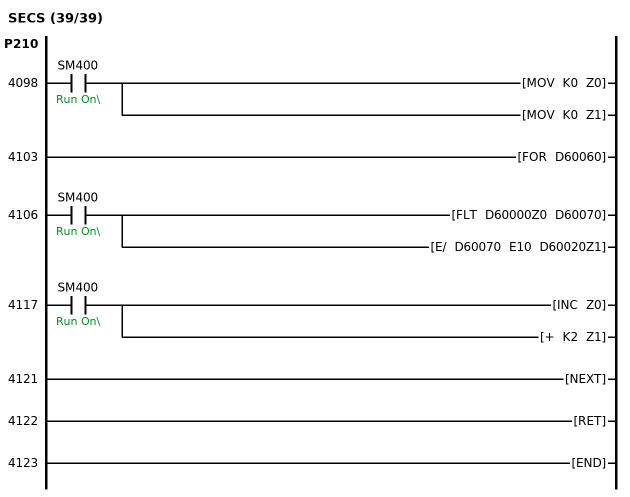
4098  LD      SM400  ; Run On\
      MOV     K0 Z0
      MOV     K0 Z1
4103  FOR     D60060
4106  LD      SM400  ; Run On\
      FLT     D60000Z0 D60070
      E/      D60070 E10 D60020Z1
4117  LD      SM400  ; Run On\
      INC     Z0
      +       K2 Z1
4121  NEXT
4122  RET
4123  END
END_PROGRAM

// device comments not shown above
D5200  ; 溫度到達H01
D5220  ; 溫度到達IRA01
D5240  ; 溫度到達IRB01
D5700  ; 低溫溫度01
D5720  ; 低溫溫度21
D20200  ; A1
D20201  ; B1
X20  ; 進料牙叉上層氣缸上定點
X21  ; 進料牙叉上層氣缸下定點
X22  ; 進料牙叉下層氣缸上定點
X23  ; 進料牙叉下層氣缸下定點
X24  ; 進料牙叉夾板氣缸開定點
X25  ; 進料牙叉夾板氣缸夾定點
X26  ; 進料牙叉左光纖檢知
X27  ; 進料牙叉右光纖檢知
X28  ; 進料吸板真空檢知
X29  ; 進料鼓風機異常
X2A  ; 進料無塵風機異常
X2D  ; 連線_上游出板要求(備用)
X2E  ; 連線_上游出板完成(備用)
X2F  ; 連線_上游備用
X30  ; 進料手臂外氣缸伸出定點
X31  ; 進料手臂外氣缸縮回定點
X32  ; 進料手臂內氣缸伸出定點
X33  ; 進料手臂內氣缸縮回定點
X34  ; 進料手臂上夾板氣缸開定點
X35  ; 進料手臂上夾板氣缸夾定點
X36  ; 進料手臂下夾板氣缸開定點
X37  ; 進料手臂下夾板氣缸夾定點
X38  ; 進料手臂右上有板檢知
X39  ; 進料手臂左上有板檢知
X3A  ; 進料手臂右下有板檢知
X3B  ; 進料手臂左下有板檢知
X3C  ; 進料安全門開關
X3D  ; 進料緊急停止開關
X3E  ; 進/出料蜂鳴器靜音按鈕
X3F  ; 進料氣源壓力檢知
X40  ; 進料回流滿框光電
X41  ; 進料回流檔框1光電
X42  ; 進料回流檔框2光電
X43  ; 進料回流檔框定點光電
X44  ; 進料檔框1氣缸D1上定點
X45  ; 進料檔框1氣缸D1下定點
X46  ; 進料檔框2氣缸D2上定點
X47  ; 進料檔框2氣缸D2下定點
X48  ; 進料後拍框氣缸A13伸出定點
X49  ; 進料後拍框氣缸A13縮回定點
X4A  ; 進料托框氣缸A12上定點
X4B  ; 進料托框氣缸A12下定點
X4C  ; 進料托伸縮氣缸A11A/B伸出定點
X4D  ; 進料托伸縮氣缸A11A/B縮回定點
X4E  ; 進料托框左光電
X4F  ; 進料托框右光電
X50  ; 進料夾框A桿前520光纖
X51  ; 進料夾框A桿前500光纖
X52  ; 進料夾框A桿前260光纖
X53  ; 進料夾框A桿前250光纖
X54  ; 進料夾框B桿前250光纖
X55  ; 進料夾框B桿前260光纖
X56  ; 進料夾框B桿前500光纖
X57  ; 進料夾框B桿前520光纖
X58  ; 進料夾框A桿後520光纖
X59  ; 進料夾框A桿後500光纖
X5A  ; 進料夾框A桿後260光纖
X5B  ; 進料夾框A桿後250光纖
X5C  ; 進料夾框B桿後250光纖
X5D  ; 進料夾框B桿後260光纖
X5E  ; 進料夾框B桿後500光纖
X5F  ; 進料夾框B桿後520光纖
X60  ; 進料左上下夾氣缸A1A/B伸出定點
X61  ; 進料左上下夾氣缸A1A/B縮回定點
X62  ; 進料左拍框氣缸A2伸出定點
X63  ; 進料左拍框氣缸A2縮回定點
X64  ; 進料左背檔框氣缸A3伸出定點
X65  ; 進料左背檔框氣缸A3縮回定點
X66  ; 進料左開爪氣缸A4伸出定點
X67  ; 進料左開爪氣缸A4縮回定點
X68  ; 進料左開框氣缸A5A/B伸出定點
X69  ; 進料左開框氣缸A5A/B縮回定點
X6A  ; 進料左上夾框光電
X6B  ; 進料左上開夾定點光纖
X6C  ; 進料左下開夾定點光纖
X6E  ; 進料左門磁簧開關
X70  ; 進料右上下夾氣缸A1A/B伸出定點
X71  ; 進料右上下夾氣缸A1A/B縮回定點
X72  ; 進料右拍框氣缸A2伸出定點
X73  ; 進料右拍框氣缸A2縮回定點
X74  ; 進料右背檔框氣缸A3伸出定點
X75  ; 進料右背檔框氣缸A3縮回定點
X76  ; 進料右開爪氣缸A4伸出定點
X77  ; 進料右開爪氣缸A4縮回定點
X78  ; 進料右開框氣缸A5A/B伸出定點
X79  ; 進料右開框氣缸A5A/B縮回定點
X7A  ; 進料右上夾框光電
X7B  ; 進料右上開夾定點光纖
X7C  ; 進料右下開夾定點光纖
X7E  ; 進料右門磁簧開關
X80  ; 分流左_伸出氣缸伸出定點
X81  ; 分流左_伸出氣缸縮回定點
X82  ; 分流左_上昇氣缸上定點
X83  ; 分流左_上昇氣缸下定點
X84  ; 分流左_框架上定點光電
X85  ; 分流左_框架下定點光電
X86  ; 分流左_旋轉定點光電
X88  ; 分流右_伸出氣缸伸出定點
X89  ; 分流右_伸出氣缸縮回定點
X8A  ; 分流右_上昇氣缸上定點
X8B  ; 分流右_上昇氣缸下定點
X8C  ; 分流右_框架上定點光電
X8D  ; 分流右_框架下定點光電
X8E  ; 分流右_旋轉定點光電
X90  ; 左IR輸送進框補助氣缸伸出定點
X91  ; 左IR輸送進框補助氣缸縮回定點
X92  ; 左IR輸送進框定位光纖
X93  ; 左IR輸送入口框架光纖
X94  ; 進料輸送排氣風車異常
X95  ; 出料輸送排氣風車異常
X98  ; 右IR輸送進框補助氣缸伸出定點
X99  ; 右IR輸送進框補助氣缸縮回定點
X9A  ; 右IR輸送進框定位光纖
X9B  ; 右IR輸送入口框架光纖
X9C  ; 進料輸送INV-A11運轉
X9D  ; 回流1輸送INV-A1運轉
X9E  ; 回流2輸送INV-A2運轉
X9F  ; 進料分流旋臂馬達INV-A3運轉
X0A0  ; 左IR輸送出框補助氣缸伸出定點
X0A1  ; 左IR輸送出框補助氣缸縮回定點
X0A2  ; 左IR輸送出口框架光纖
X0A3  ; 左IR輸送出框定位光纖
X0A4  ; 左IR輸送出框定點光纖
X0A5  ; 左IR輸送拉框氣缸伸出定點
X0A6  ; 左IR輸送拉框氣缸縮回定點
X0A7  ; 左IR輸送勾框氣缸伸出定點
X0A8  ; 右IR輸送出框補助氣缸伸出定點
X0A9  ; 右IR輸送出框補助氣缸縮回定點
X0AA  ; 右IR輸送出口框架光纖
X0AB  ; 右IR輸送出框定位光纖
X0AC  ; 右IR輸送出框定點光纖
X0AD  ; 右IR輸送拉框氣缸伸出定點
X0AE  ; 右IR輸送拉框氣缸縮回定點
X0AF  ; 右IR輸送勾框氣缸伸出定點
X0B0  ; 合流左_伸出氣缸伸出定點
X0B1  ; 合流左_伸出氣缸縮回定點
X0B2  ; 合流左_上昇氣缸上定點
X0B3  ; 合流左_上昇氣缸下定點
X0B4  ; 合流左_框架上定點光電
X0B5  ; 合流左_框架下定點光電
X0B6  ; 合流左_旋轉定點光電
X0B8  ; 合流右_伸出氣缸伸出定點
X0B9  ; 合流右_伸出氣缸縮回定點
X0BA  ; 合流右_上昇氣缸上定點
X0BB  ; 合流右_上昇氣缸下定點
X0BC  ; 合流右_框架上定點光電
X0BD  ; 合流右_框架下定點光電
X0BE  ; 合流右_旋轉定點光電
X0C0  ; 出料左上下夾氣缸B01A/B伸出定點
X0C1  ; 出料左上下夾氣缸B01A/B縮回定點
X0C2  ; 出料左拍框氣缸B02伸出定點
X0C3  ; 出料左拍框氣缸B02縮回定點
X0C4  ; 出料左背檔框氣缸B03伸出定點
X0C5  ; 出料左背檔框氣缸B03縮回定點
X0C6  ; 出料左開爪氣缸B04伸出定點
X0C7  ; 出料左開爪氣缸B04縮回定點
X0C8  ; 出料左開框氣缸B05A/B伸出定點
X0C9  ; 出料左開框氣缸B05A/B縮回定點
X0CA  ; 出料左上夾框光電
X0CB  ; 出料左上開夾定點光纖
X0CC  ; 出料左下開夾定點光纖
X0CD  ; 出料左無板確認光電
X0CE  ; 出料左門磁簧開關
X0D0  ; 出料右上下夾氣缸B01A/B伸出定點
X0D1  ; 出料右上下夾氣缸B01A/B縮回定點
X0D2  ; 出料右拍框氣缸B02伸出定點
X0D3  ; 出料右拍框氣缸B02縮回定點
X0D4  ; 出料右背檔框氣缸B03伸出定點
X0D5  ; 出料右背檔框氣缸B03縮回定點
X0D6  ; 出料右開爪氣缸B04伸出定點
X0D7  ; 出料右開爪氣缸B04縮回定點
X0D8  ; 出料右開框氣缸B05A/B伸出定點
X0D9  ; 出料右開框氣缸B05A/B縮回定點
X0DA  ; 出料右上夾框光電
X0DB  ; 出料右上開夾定點光纖
X0DC  ; 出料右下開夾定點光纖
X0DD  ; 出料右無板確認光電
X0DE  ; 出料右門磁簧開關
X0E0  ; 出料回流滿框光電
X0E1  ; 出料回流框架檢知光電
X0E2  ; 出料回流框架脫離光電
X0E6  ; 出料下導框氣缸B14伸出定點
X0E7  ; 出料下導框氣缸B14縮回定點
X0E8  ; 出料推框氣缸B13伸出定點
X0E9  ; 出料推框氣缸B13縮回定點
X0EA  ; 出料托框氣缸B12上定點
X0EB  ; 出料托框氣缸B12下一定點
X0EC  ; 出料托框伸縮氣缸B11A/B伸出定點
X0ED  ; 出料托框伸縮氣缸B11A/B縮回定點
X0EE  ; 出料托框左光電
X0EF  ; 出料托框右光電
X0F0  ; 出料手臂外氣缸伸出定點
X0F1  ; 出料手臂外氣缸縮回定點
X0F2  ; 出料手臂內氣缸伸出定點
X0F3  ; 出料手臂內氣缸縮回定點
X0F4  ; 出料手臂上夾板氣缸開定點
X0F5  ; 出料手臂上夾板氣缸夾定點
X0F6  ; 出料手臂下夾板氣缸開定點
X0F7  ; 出料手臂下夾板氣缸夾定點
X0F8  ; 出料手臂右上有板檢知
X0F9  ; 出料手臂左上有板檢知
X0FA  ; 出料手臂右下有板檢知
X0FB  ; 出料手臂左下有板檢知
X0FC  ; 出料安全門開關
X0FD  ; 出料緊急停止開關
X0FE  ; 電源相序檢知
X0FF  ; 出料氣源壓力檢知
X104  ; 出料平台頂昇氣缸上定點
X105  ; 出料平台頂昇氣缸下定點
X106  ; 出料輸送左側光電
X107  ; 出料輸送右側光電
X108  ; 出料輸送入口光電
X109  ; 出料無塵風機異常
X10A  ; 出料旋臂馬達INV-C01運轉
X10B  ; 出料旋臂馬達INV-C02運轉
X10D  ; 連線_下游允許出板
X10E  ; 連線_下游出板中(備用)
X110  ; 左冷卻排氣風車異常
X111  ; 左冷卻無塵風機異常
X112  ; 左IR輸送INV-B01運轉
X118  ; 右冷卻排氣風車異常
X119  ; 右冷卻無塵風機異常
X11A  ; 右IR輸送INV-B01運轉
X11C  ; 第09槽電熱箱H09超溫防止器
X11D  ; 第10槽電熱箱H10超溫防止器
X11E  ; 第11槽電熱箱H11超溫防止器
X11F  ; 第12槽電熱箱H12超溫防止器
X120  ; 第01槽風車馬達過載異常
X121  ; 第02槽風車馬達過載異常
X122  ; 第03槽風車馬達過載異常
X123  ; 第04槽風車馬達過載異常
X124  ; 第05槽風車馬達過載異常
X125  ; 第06槽風車馬達過載異常
X126  ; 第07槽風車馬達過載異常
X127  ; 第08槽風車馬達過載異常
X128  ; 第01槽風車馬達電流檢知
X129  ; 第02槽風車馬達電流檢知
X12A  ; 第03槽風車馬達電流檢知
X12B  ; 第04槽風車馬達電流檢知
X12C  ; 第05槽風車馬達電流檢知
X12D  ; 第06槽風車馬達電流檢知
X12E  ; 第07槽風車馬達電流檢知
X12F  ; 第08槽風車馬達電流檢知
X130  ; 第01槽電熱箱H01超溫防止器
X131  ; 第02槽電熱箱H02超溫防止器
X132  ; 第03槽電熱箱H03超溫防止器
X133  ; 第04槽電熱箱H04超溫防止器
X134  ; 第05槽電熱箱H05超溫防止器
X135  ; 第06槽電熱箱H06超溫防止器
X136  ; 第07槽電熱箱H07超溫防止器
X137  ; 第08槽電熱箱H08超溫防止器
X138  ; 第01槽IR01A超溫防止器
X139  ; 第02槽IR02A超溫防止器
X13A  ; 第03槽IR03A超溫防止器
X13B  ; 第04槽IR04A超溫防止器
X13C  ; 第05槽IR05A超溫防止器
X13D  ; 第06槽IR06A超溫防止器
X13E  ; 第07槽IR07A超溫防止器
X13F  ; 第08槽IR08A超溫防止器
X140  ; 第01槽熱風H01溫度到達
X141  ; 第02槽熱風H02溫度到達
X142  ; 第03槽熱風H03溫度到達
X143  ; 第04槽熱風H04溫度到達
X144  ; 第05槽熱風H05溫度到達
X145  ; 第06槽熱風H06溫度到達
X146  ; 第07槽熱風H07溫度到達
X147  ; 第08槽熱風H08溫度到達
X148  ; 第01槽IR01A溫度到達
X149  ; 第02槽IR02A溫度到達
X14A  ; 第03槽IR03A溫度到達
X14B  ; 第04槽IR04A溫度到達
X14C  ; 第05槽IR05A溫度到達
X14D  ; 第06槽IR06A溫度到達
X14E  ; 第07槽IR07A溫度到達
X14F  ; 第08槽IR08A溫度到達
X150  ; 第01槽H01溫控超溫異常
X151  ; 第02槽H02溫控超溫異常
X152  ; 第03槽H03溫控超溫異常
X153  ; 第04槽H04溫控超溫異常
X154  ; 第05槽H05溫控超溫異常
X155  ; 第06槽H06溫控超溫異常
X156  ; 第07槽H07溫控超溫異常
X157  ; 第08槽H08溫控超溫異常
X158  ; 第01槽IR01A溫控超溫異常
X159  ; 第02槽IR02A溫控超溫異常
X15A  ; 第03槽IR03A溫控超溫異常
X15B  ; 第04槽IR04A溫控超溫異常
X15C  ; 第05槽IR05A溫控超溫異常
X15D  ; 第06槽IR06A溫控超溫異常
X15E  ; 第07槽IR07A溫控超溫異常
X15F  ; 第08槽IR08A溫控超溫異常
X160  ; 第09槽風車馬達過載異常
X161  ; 第10槽風車馬達過載異常
X162  ; 第11槽風車馬達過載異常
X163  ; 第12槽風車馬達過載異常
X164  ; 第09槽風車馬達電流檢知
X165  ; 第10槽風車馬達電流檢知
X166  ; 第11槽風車馬達電流檢知
X167  ; 第12槽風車馬達電流檢知
X168  ; 第09槽SCR09/09A/09B異常
X169  ; 第10槽SCR10/10A/10B異常
X16A  ; 第11槽SCR11/911/11B異常
X16B  ; 第12槽SCR12/12A/12B異常
X16C  ; 第09槽分路開關跳脫異常
X16D  ; 第10槽分路開關跳脫異常
X16E  ; 第11槽分路開關跳脫異常
X16F  ; 第12槽分路開關跳脫異常
X170  ; 第01槽SCR01/01A/01B異常
X171  ; 第02槽SCR02/02A/02B異常
X172  ; 第03槽SCR03/03A/03B異常
X173  ; 第04槽SCR04/04A/04B異常
X174  ; 第05槽SCR05/05A/05B異常
X175  ; 第06槽SCR06/06A/06B異常
X176  ; 第07槽SCR07/07A/07B異常
X177  ; 第08槽SCR08/08A/08B異常
X178  ; 第01槽分路開關跳脫異常
X179  ; 第02槽分路開關跳脫異常
X17A  ; 第03槽分路開關跳脫異常
X17B  ; 第04槽分路開關跳脫異常
X17C  ; 第05槽分路開關跳脫異常
X17D  ; 第06槽分路開關跳脫異常
X17E  ; 第07槽分路開關跳脫異常
X17F  ; 第08槽分路開關跳脫異常
X180  ; 第01槽IR01B溫度到達
X181  ; 第02槽IR02B溫度到達
X182  ; 第03槽IR03B溫度到達
X183  ; 第04槽IR04B溫度到達
X184  ; 第05槽IR05B溫度到達
X185  ; 第06槽IR06B溫度到達
X186  ; 第07槽IR07B溫度到達
X187  ; 第08槽IR08B溫度到達
X188  ; 第01槽IR01B溫控超溫異常
X189  ; 第02槽IR02B溫控超溫異常
X18A  ; 第03槽IR03B溫控超溫異常
X18B  ; 第04槽IR04B溫控超溫異常
X18C  ; 第05槽IR05B溫控超溫異常
X18D  ; 第06槽IR06B溫控超溫異常
X18E  ; 第07槽IR07B溫控超溫異常
X18F  ; 第08槽IR08B溫控超溫異常
X190  ; 第01槽IR01B超溫防止器
X191  ; 第02槽IR02B超溫防止器
X192  ; 第03槽IR03B超溫防止器
X193  ; 第04槽IR04B超溫防止器
X194  ; 第05槽IR05B超溫防止器
X195  ; 第06槽IR06B超溫防止器
X196  ; 第07槽IR07B超溫防止器
X197  ; 第08槽IR08B超溫防止器
X198  ; 第09槽IR09A超溫防止器
X199  ; 第10槽IR10A超溫防止器
X19A  ; 第11槽IR11A超溫防止器
X19B  ; 第12槽IR12A超溫防止器
X19C  ; 第09槽IR09B超溫防止器
X19D  ; 第10槽IR10B超溫防止器
X19E  ; 第11槽IR11B超溫防止器
X19F  ; 第12槽IR12B超溫防止器
X1A0  ; 第09槽熱風H09溫度到達
X1A1  ; 第09槽H09溫控超溫異常
X1A2  ; 第09槽IR09A溫度到達
X1A3  ; 第09槽IR09A溫控超溫異常
X1A4  ; 第09槽IR09B溫度到達
X1A5  ; 第09槽IR09B溫控超溫異常
X1A8  ; 第10槽熱風H10溫度到達
X1A9  ; 第10槽H10溫控超溫異常
X1AA  ; 第10槽IR10A溫度到達
X1AB  ; 第10槽IR10A溫控超溫異常
X1AC  ; 第10槽IR10B溫度到達
X1AD  ; 第10槽IR10B溫控超溫異常
X1B0  ; 第11槽熱風H11溫度到達
X1B1  ; 第11槽H11溫控超溫異常
X1B2  ; 第11槽IR11A溫度到達
X1B3  ; 第11槽IR11A溫控超溫異常
X1B4  ; 第11槽IR11B溫度到達
X1B5  ; 第11槽IR11B溫控超溫異常
X1B8  ; 第12槽熱風H12溫度到達
X1B9  ; 第12槽H12溫控超溫異常
X1BA  ; 第12槽IR12A溫度到達
X1BB  ; 第12槽IR12A溫控超溫異常
X1BC  ; 第12槽IR12B溫度到達
X1BD  ; 第12槽IR12B溫控超溫異常
X0A23  ; Other station   DataLinkStatus
X0A48  ; High resolutuon mode status flag
X0A49  ; Operating condition setting ok
X0A4A  ; Offset/gain setting mode flag
X0A4B  ; Channel change completed flag
X0A4C  ; Set value change completed flag
X0A4D  ; Synchronous mode flag
X1007  ; 進料手臂_(DO08)
X1008  ; 進料手臂_(DO09)
X1009  ; 進料手臂_AB放板#3位置(DO10)
X100D  ; 進料手臂_(DO14)
X1010  ; 進料手臂_(DO17)
X1011  ; 進料手臂_(DO18)
X1012  ; 進料手臂_(DO19)
X1013  ; 進料手臂_(DO20)
X1014  ; 進料手臂_(DO21)
X1015  ; 進料手臂_(DO22)
X1016  ; 進料手臂_(DO23)
X1018  ; 進料手臂_(DO25)
X1019  ; 進料手臂_(DO26)
X101D  ; 進料手臂_(DO30)
X101E  ; 進料手臂_(DO31)
X101F  ; 進料手臂_(DO32)
X1024  ; 進料手臂_CCD再校正一次OK(DO37)
X1026  ; 進料手臂_原點往X軸移動-20MM(DO39
X1027  ; 進料手臂_原點往Y軸移動-20MM(DO40
X1028  ; 進料手臂_原點往T軸正轉移動2度(DO
X1029  ; 進料手臂_(DO42)
X102C  ; 進料手臂_B放板完成位置(DO45)
X102E  ; 進料手臂_(DO47)
X102F  ; 進料手臂_(DO48)
X1030  ; 進料手臂_(DO49)
X1031  ; 進料手臂_(DO50)
X1032  ; 進料手臂_(DO51)
X1033  ; 進料手臂_(DO52)
X1034  ; 進料手臂_(DO53)
X1035  ; 進料手臂_(DO54)
X1036  ; 進料手臂_(DO55)
X1037  ; 進料手臂_(DO56)
X1038  ; 進料手臂_(DO57)
X1039  ; 進料手臂_(DO58)
X103A  ; 進料手臂_(DO59)
X103B  ; 進料手臂_(DO60)
X103C  ; 進料手臂_(DO61)
X103D  ; 進料手臂_(DO62)
X103E  ; 進料手臂_(DO63)
X103F  ; 進料手臂_(DO64)
X1040  ; 進料手臂_放板位置_P32-3(DO65)
X1041  ; 進料手臂_放板位置_P32-2(DO66)
X1042  ; 進料手臂_放板位置_P32-1(DO67)
X1043  ; 進料手臂_放板完成位置_P33-10(DO6
X1044  ; 進料手臂_放板完成位置_P33-9(DO69
X1045  ; 進料手臂_(DO70)
X1046  ; 進料手臂_(DO71)
X1047  ; 進料手臂_(DO72)
X1048  ; 進料手臂_(DO73)
X1049  ; 進料手臂_(DO74)
X104A  ; 進料手臂_(DO75)
X104B  ; 進料手臂_(DO76)
X104C  ; 進料手臂_(DO77)
X104D  ; 進料手臂_(DO78)
X104E  ; 進料手臂_(DO79)
X104F  ; 進料手臂_(DO80)
X1050  ; 進料手臂_(DO81)
X1051  ; 進料手臂_(DO82)
X1052  ; 進料手臂_(DO83)
X1053  ; 進料手臂_(DO84)
X1054  ; 進料手臂_(DO85)
X1055  ; 進料手臂_(DO86)
X1056  ; 進料手臂_(DO87)
X1057  ; 進料手臂_(DO88)
X1058  ; 進料手臂_(DO89)
X1059  ; 進料手臂_(DO90)
X105A  ; 進料手臂_(DO91)
X105B  ; 進料手臂_(DO92)
X105C  ; 進料手臂_(DO93)
X105D  ; 進料手臂_(DO94)
X105E  ; 進料手臂_(DO95)
X105F  ; 進料手臂_(DO96)
X1060  ; 進料手臂_(DO97)
X1061  ; 進料手臂_(DO98)
X1062  ; 進料手臂_(DO99)
X1063  ; 進料手臂_(DO100)
X1064  ; 進料手臂_(DO101)
X1065  ; 進料手臂_(DO102)
X1066  ; 進料手臂_(DO103)
X1067  ; 進料手臂_(DO104)
X1068  ; 進料手臂_(DO105)
X1069  ; 進料手臂_(DO106)
X106A  ; 進料手臂_(DO107)
X106B  ; 進料手臂_(DO108)
X106C  ; 進料手臂_(DO109)
X106D  ; 進料手臂_(DO110)
X106E  ; 進料手臂_(DO111)
X106F  ; 進料手臂_(DO112)
X1070  ; 進料手臂_(DO113)
X1071  ; 進料手臂_(DO114)
X1072  ; 進料手臂_(DO115)
X1073  ; 進料手臂_(DO116)
X1074  ; 進料手臂_(DO117)
X1075  ; 進料手臂_(DO118)
X1076  ; 進料手臂_(DO119)
X1077  ; 進料手臂_(DO120)
X1078  ; 進料手臂_(DO121)
X1079  ; 進料手臂_(DO122)
X107A  ; 進料手臂_(DO123)
X107B  ; 進料手臂_(DO124)
X107C  ; 進料手臂_(DO125)
X107D  ; 進料手臂_(DO126)
X107E  ; 進料手臂_(DO127)
X107F  ; 進料手臂_(DO128)
X1087  ; 出料手臂_(DO08)
X1088  ; 出料手臂_(DO09)
X1089  ; 出料手臂_AB放板#3位置(DO10)
X108D  ; 出料手臂_(DO14)
X1090  ; 出料手臂_(DO17)
X1091  ; 出料手臂_(DO18)
X1092  ; 出料手臂_(DO19)
X1093  ; 出料手臂_(DO20)
X1094  ; 出料手臂_(DO21)
X1095  ; 出料手臂_(DO22)
X1096  ; 出料手臂_(DO23)
X1098  ; 出料手臂_(DO25)
X1099  ; 出料手臂_(DO26)
X109D  ; 出料手臂_(DO30)
X109E  ; 出料手臂_(DO31)
X109F  ; 出料手臂_(DO32)
X10A0  ; 出料手臂_Y+20-OK(DO33)
X10A1  ; 出料手臂_X+20-OK(DO34)
X10A2  ; 出料手臂_Y-20-OK(DO35)
X10A3  ; 出料手臂_X-20-OK(DO36)
X10A4  ; 出料手臂_CCD再校正一次OK(DO37)
X10A5  ; 出料手臂_校正位置OK(DO38)
X10A6  ; 出料手臂_原點往X軸移動-20MM(DO39
X10A7  ; 出料手臂_原點往Y軸移動-20MM(DO40
X10A8  ; 出料手臂_原點往T軸正轉移動2度
X10A9  ; 出料手臂_(DO42)
X10AA  ; 出料手臂_(DO43)
X10AB  ; 出料手臂_B放板上升位置(DO44)
X10AC  ; 出料手臂_B放板完成位置(DO45)
X10AD  ; 出料手臂_T180-OK(DO46)
X10AE  ; 出料手臂_(DO47)
X10AF  ; 出料手臂_(DO48)
X10B0  ; 出料手臂_(DO49)
X10B1  ; 出料手臂_(DO50)
X10B2  ; 出料手臂_(DO51)
X10B3  ; 出料手臂_(DO52)
X10B4  ; 出料手臂_(DO53)
X10B5  ; 出料手臂_(DO54)
X10B6  ; 出料手臂_(DO55)
X10B7  ; 出料手臂_(DO56)
X10B8  ; 出料手臂_(DO57)
X10B9  ; 出料手臂_(DO58)
X10BA  ; 出料手臂_(DO59)
X10BB  ; 出料手臂_(DO60)
X10BC  ; 出料手臂_(DO61)
X10BD  ; 出料手臂_(DO62)
X10BE  ; 出料手臂_(DO63)
X10BF  ; 出料手臂_(DO64)
X10C0  ; 出料手臂_放板位置_P32-3(DO65)
X10C1  ; 出料手臂_放板位置_P32-2(DO66)
X10C2  ; 出料手臂_放板位置_P32-1(DO67)
X10C3  ; 出料手臂_放板完成位置_P33-10(DO6
X10C4  ; 出料手臂_放板完成位置_P33-9(DO69
X10C5  ; 出料手臂_(DO70)
X10C6  ; 出料手臂_(DO71)
X10C7  ; 出料手臂_(DO72)
X10C8  ; 出料手臂_(DO73)
X10C9  ; 出料手臂_(DO74)
X10CA  ; 出料手臂_(DO75)
X10CB  ; 出料手臂_(DO76)
X10CC  ; 出料手臂_(DO77)
X10CD  ; 出料手臂_(DO78)
X10CE  ; 出料手臂_(DO79)
X10CF  ; 出料手臂_(DO80)
X10D0  ; 出料手臂_(DO81)
X10D1  ; 出料手臂_(DO82)
X10D2  ; 出料手臂_(DO83)
X10D3  ; 出料手臂_(DO84)
X10D4  ; 出料手臂_(DO85)
X10D5  ; 出料手臂_(DO86)
X10D6  ; 出料手臂_(DO87)
X10D7  ; 出料手臂_(DO88)
X10D8  ; 出料手臂_(DO89)
X10D9  ; 出料手臂_(DO90)
X10DA  ; 出料手臂_(DO91)
X10DB  ; 出料手臂_(DO92)
X10DC  ; 出料手臂_(DO93)
X10DD  ; 出料手臂_(DO94)
X10DE  ; 出料手臂_(DO95)
X10DF  ; 出料手臂_(DO96)
X10E0  ; 出料手臂_(DO97)
X10E1  ; 出料手臂_(DO98)
X10E2  ; 出料手臂_(DO99)
X10E3  ; 出料手臂_(DO100)
X10E4  ; 出料手臂_(DO101)
X10E5  ; 出料手臂_(DO102)
X10E6  ; 出料手臂_(DO103)
X10E7  ; 出料手臂_(DO104)
X10E8  ; 出料手臂_(DO105)
X10E9  ; 出料手臂_(DO106)
X10EA  ; 出料手臂_(DO107)
X10EB  ; 出料手臂_(DO108)
X10EC  ; 出料手臂_(DO109)
X10ED  ; 出料手臂_(DO110)
X10EE  ; 出料手臂_(DO111)
X10EF  ; 出料手臂_(DO112)
X10F0  ; 出料手臂_(DO113)
X10F1  ; 出料手臂_(DO114)
X10F2  ; 出料手臂_(DO115)
X10F3  ; 出料手臂_(DO116)
X10F4  ; 出料手臂_(DO117)
X10F5  ; 出料手臂_(DO118)
X10F6  ; 出料手臂_(DO119)
X10F7  ; 出料手臂_(DO120)
X10F8  ; 出料手臂_(DO121)
X10F9  ; 出料手臂_(DO122)
X10FA  ; 出料手臂_(DO123)
X10FB  ; 出料手臂_(DO124)
X10FC  ; 出料手臂_(DO125)
X10FD  ; 出料手臂_(DO126)
X10FE  ; 出料手臂_(DO127)
X10FF  ; 出料手臂_(DO128)
Y200  ; 進料牙叉上層氣缸A20上昇SV
Y201  ; 進料牙叉上層氣缸A20下降SV
Y202  ; 進料牙叉下層氣缸A21上昇SV
Y203  ; 進料牙叉下層氣缸A21下降SV
Y204  ; 進料牙叉夾板氣缸A22伸出SV
Y205  ; 進料牙叉夾板氣缸A22縮回SV
Y206  ; 進料真空氣缸A23吸板SV
Y207  ; 進料真空氣缸A23放板SV
Y208  ; 進料真空外側分區A24SV
Y209  ; 進料真空外側分區A25SV
Y20A  ; 進料鼓風機電磁開關
Y20B  ; 進/出料蜂鳴器
Y20C  ; 進/出料三色燈藍燈
Y20D  ; 進/出料三色燈綠燈
Y20E  ; 進/出料三色燈黃燈
Y20F  ; 進/出料三色燈紅燈
Y210  ; 進料手臂板寬氣缸A30伸出SV
Y211  ; 進料手臂板寬氣缸A30縮回SV
Y212  ; 進料手臂上夾板氣缸A31夾板SV
Y213  ; 進料手臂下夾板氣缸A32夾板SV
Y214  ; 進料檔框1氣缸D1伸出SV
Y215  ; 進料檔框1氣缸D1縮回SV
Y216  ; 進料檔框2氣缸D2伸出SV
Y217  ; 進料檔框2氣缸D2縮回SV
Y218  ; 進料後拍框氣缸A13伸出SV
Y219  ; 進料後拍框氣缸A13縮回SV
Y21A  ; 進料托架氣缸A12上昇SV
Y21B  ; 進料托架氣缸A12下降SV
Y21C  ; 進料托框伸縮氣缸伸出SV
Y21D  ; 進料托框伸縮氣缸縮回SV
Y21E  ; CCD照明繼電器
Y220  ; 進料左上下夾框氣缸A1A/B伸出SV
Y221  ; 進料左上下夾框氣缸A1A/B縮回SV
Y222  ; 進料左拍框氣缸A2伸出SV
Y223  ; 進料左拍框氣缸A2縮回SV
Y224  ; 進料左背檔框氣缸A3伸出SV
Y225  ; 進料左背檔框氣缸A3縮回SV
Y226  ; 進料左開爪氣缸A4伸出SV
Y227  ; 進料左開爪氣缸A4縮回SV
Y228  ; 進料左開框氣缸A5A/B伸出SV
Y229  ; 進料左開框氣缸A5A/B縮回SV
Y22D  ; 上游_允許進板訊號
Y22E  ; 上游_進板中訊號
Y22F  ; 上游_啟動完成訊號
Y230  ; 進料右上下夾框氣缸A6A/B伸出SV
Y231  ; 進料右上下夾框氣缸A6A/B縮回SV
Y232  ; 進料右拍框氣缸A7伸出SV
Y233  ; 進料右拍框氣缸A7縮回SV
Y234  ; 進料右背檔框氣缸A8伸出SV
Y235  ; 進料右背檔框氣缸A8縮回SV
Y236  ; 進料右開爪氣缸A9伸出SV
Y237  ; 進料右開爪氣缸A9縮回SV
Y238  ; 進料右開框氣缸A10A/B伸出SV
Y239  ; 進料右開框氣缸A10A/B縮回SV
Y240  ; 分流左_伸出氣缸C1伸出SV
Y241  ; 分流左_伸出氣缸C1縮回SV
Y242  ; 分流左_上昇氣缸C2上昇SV
Y243  ; 分流左_下降氣缸C2下降SV
Y244  ; 左IR輸送進框補助氣缸C3伸出SV
Y245  ; 左IR輸送進框補助氣缸C3縮回SV
Y246  ; 分流右_伸出氣缸C4伸出SV
Y247  ; 分流右_伸出氣缸C4縮回SV
Y248  ; 分流右_上昇氣缸C5上昇SV
Y249  ; 分流右_下降氣缸C5下降SV
Y24A  ; 右IR輸送進框補助氣缸C6伸出SV
Y24B  ; 右IR輸送進框補助氣缸C6縮回SV
Y24C  ; 框架回流輸送1變頻器INVA1運轉
Y24D  ; 框架回流輸送2變頻器INVA2運轉
Y24E  ; 進料分流旋臂變頻器INVA3運轉
Y24F  ; 進料變頻器異常復歸
Y260  ; 合流左_伸出氣缸C11伸出SV
Y261  ; 合流左_伸出氣缸C11縮回SV
Y262  ; 合流左_上昇氣缸C12上昇SV
Y263  ; 合流左_下降氣缸C12下降SV
Y264  ; 左IR輸送出框補助氣缸C13伸出SV
Y265  ; 左IR輸送出框補助氣缸C13縮回SV
Y266  ; 合流右_伸出氣缸C14伸出SV
Y267  ; 合流右_伸出氣缸C14縮回SV
Y268  ; 合流右_上昇氣缸C15上昇SV
Y269  ; 合流右_下降氣缸C15下降SV
Y26A  ; 右IR輸送出框補助氣缸C16伸出SV
Y26B  ; 右IR輸送出框補助氣缸C16縮回SV
Y26C  ; 左IR輸送變頻器INVB1運轉
Y26D  ; 右IR輸送變頻器INVB2運轉
Y26E  ; 出料合流旋臂變頻器INVC1運轉
Y26F  ; 出料變頻器異常復歸
Y270  ; 出料左上下夾框氣缸B1A/B伸出SV
Y271  ; 出料左上下夾框氣缸B1A/B縮回SV
Y272  ; 出料左拍框氣缸B2伸出SV
Y273  ; 出料左拍框氣缸B2縮回SV
Y274  ; 出料左背檔框氣缸B3伸出SV
Y275  ; 出料左背檔框氣缸B3縮回SV
Y276  ; 出料左開爪氣缸B4伸出SV
Y277  ; 出料左開爪氣缸B4縮回SV
Y278  ; 出料左開框氣缸B5A/B伸出SV
Y279  ; 出料左開框氣缸B5A/B縮回SV
Y27A  ; 左IR輸送拉框氣缸C14伸出SV
Y27B  ; 左IR輸送拉框氣缸C14縮回SV
Y27C  ; 左IR輸送勾框氣缸C15伸出SV
Y27D  ; 右IR輸送拉框氣缸C24伸出SV
Y27E  ; 右IR輸送拉框氣缸C24縮回SV
Y27F  ; 右IR輸送勾框氣缸C25伸出SV
Y280  ; 出料右上下夾框氣缸B6A/B伸出SV
Y281  ; 出料右上下夾框氣缸B6A/B縮回SV
Y282  ; 出料右拍框氣缸B7伸出SV
Y283  ; 出料右拍框氣缸B7縮回SV
Y284  ; 出料右背檔框氣缸B8伸出SV
Y285  ; 出料右背檔框氣缸B8縮回SV
Y286  ; 出料右開爪氣缸B9伸出SV
Y287  ; 出料右開爪氣缸B9縮回SV
Y288  ; 出料右開框氣缸B10A/B伸出SV
Y289  ; 出料右開框氣缸B10A/B縮回SV
Y28A  ; 出料平台頂昇氣缸B20上昇SV
Y28B  ; 出料平台頂昇氣缸B20下降SV
Y28D  ; 出料輸送變頻器INVC2運轉
Y28E  ; 出料輸送變頻器INVC2慢速
Y28F  ; 出料輸送變頻器異常復歸
Y290  ; 出料手臂板寬氣缸B30伸出SV
Y291  ; 出料手臂板寬氣缸B30縮回SV
Y292  ; 出料手臂上夾板氣缸B31夾板SV
Y293  ; 出料手臂下夾板氣缸B32夾板SV
Y294  ; 出料下導框氣缸B14伸出SV
Y295  ; 出料下導框氣缸B14縮回SV
Y296  ; 出料推框氣缸B12伸出SV
Y297  ; 出料推框氣缸B12縮回SV
Y298  ; 出料托架氣缸B12上昇SV
Y299  ; 出料托架氣缸B12下降SV
Y29A  ; 出料托框伸縮氣缸B11A/B伸出SV
Y29B  ; 出料托框伸縮氣缸B11A/B縮回SV
Y29D  ; 下游_出板要求訊號
Y29E  ; 下游_出板中訊號
Y29F  ; 下游_啟動完成訊號
Y2A0  ; 第01槽熱風H01電磁開關
Y2A1  ; 第02槽熱風H02電磁開關
Y2A2  ; 第03槽熱風H03電磁開關
Y2A3  ; 第04槽熱風H04電磁開關
Y2A4  ; 第05槽熱風H05電磁開關
Y2A5  ; 第06槽熱風H06電磁開關
Y2A6  ; 第07槽熱風H07電磁開關
Y2A7  ; 第08槽熱風H08電磁開關
Y2A8  ; 第01槽IR01A電磁開關
Y2A9  ; 第02槽IR02A電磁開關
Y2AA  ; 第03槽IR03A電磁開關
Y2AB  ; 第04槽IR04A電磁開關
Y2AC  ; 第05槽IR05A電磁開關
Y2AD  ; 第06槽IR06A電磁開關
Y2AE  ; 第07槽IR07A電磁開關
Y2AF  ; 第08槽IR08A電磁開關
Y2B0  ; 第01槽風車電磁開關
Y2B1  ; 第02槽風車電磁開關
Y2B2  ; 第03槽風車電磁開關
Y2B3  ; 第04槽風車電磁開關
Y2B4  ; 第05槽風車電磁開關
Y2B5  ; 第06槽風車電磁開關
Y2B6  ; 第07槽風車電磁開關
Y2B7  ; 第08槽風車電磁開關
Y2B8  ; 左冷卻排氣風車電磁開關
Y2B9  ; 右冷卻排氣風車電磁開關
Y2BA  ; 進料無塵風機電磁開關
Y2BB  ; 出料無塵風機電磁開關
Y2BC  ; 進料輸送排氣電磁開關
Y2BD  ; 出料輸送排氣電磁開關
Y2BE  ; 左冷卻FFU風機電磁開關
Y2BF  ; 右冷卻FFU風機電磁開關
Y2C0  ; 第09槽熱風H09電磁開關
Y2C1  ; 第10槽熱風H10電磁開關
Y2C2  ; 第11槽熱風H11電磁開關
Y2C3  ; 第12槽熱風H12電磁開關
Y2C8  ; 第09槽IR09A電磁開關
Y2C9  ; 第10槽IR10A電磁開關
Y2CA  ; 第11槽IR11A電磁開關
Y2CB  ; 第12槽IR12A電磁開關
Y2CC  ; 第09槽IR09B電磁開關
Y2CD  ; 第10槽IR10B電磁開關
Y2CE  ; 第11槽IR11B電磁開關
Y2CF  ; 第12槽IR12B電磁開關
Y2D0  ; 第09槽風車電磁開關
Y2D1  ; 第10槽風車電磁開關
Y2D2  ; 第11槽風車電磁開關
Y2D3  ; 第12槽風車電磁開關
Y2D8  ; 第01槽IR01B電磁開關
Y2D9  ; 第02槽IR02B電磁開關
Y2DA  ; 第03槽IR03B電磁開關
Y2DB  ; 第04槽IR04B電磁開關
Y2DC  ; 第05槽IR05B電磁開關
Y2DD  ; 第06槽IR06B電磁開關
Y2DE  ; 第07槽IR07B電磁開關
Y2DF  ; 第08槽IR08B電磁開關
Y0A19  ; #10 AXIS Start
Y0A1F  ; #16 AXIS Start
Y0A43  ; CH03 Output enable/disable flag
Y0A44  ; CH04 Output enable/disable flag
Y0A45  ; CH05 Output enable/disable flag
Y0A46  ; CH06 Output enable/disable flag
Y0A47  ; CH07 Output enable/disable flag
Y0A48  ; CH08 Output enable/disable flag
Y0A49  ; Operating condition setting requ
Y0A4A  ; User range writing request
Y0A4B  ; Channel change request
Y0A4C  ; Set value change request
Y0A4D  ; Synchronous output request
Y1007  ; 進料手臂_(DI08)
Y1008  ; 進料手臂_(DI09)
Y1009  ; 進料手臂_(DI10)
Y100D  ; 進料手臂_(DI14)
Y1011  ; 進料手臂_(DI18)
Y1012  ; 進料手臂_(DI19)
Y1013  ; 進料手臂_(DI20)
Y1015  ; 進料手臂_(DI22)
Y1016  ; 進料手臂_(DI23)
Y1017  ; 進料手臂_(DI24)
Y1018  ; 進料手臂_(DI25)
Y1019  ; 進料手臂_(DI26)
Y101D  ; 進料手臂_(DI30)
Y101E  ; 進料手臂_(DI31)
Y101F  ; 進料手臂_(DI32)
Y1024  ; 進料手臂_CCD再校正一次(DI37)
Y1026  ; 進料手臂_原點往X軸移動-20MM(DI39
Y1027  ; 進料手臂_原點往Y軸移動-20MM(DI40
Y1028  ; 進料手臂_原點往T軸正轉移動2度(DI
Y1029  ; 進料手臂_(DI42)
Y102A  ; 進料手臂_B放板待命位置(DI43)
Y102B  ; 進料手臂_B放板上升位置(DI44)
Y102C  ; 進料手臂_B放板完成位置(DI45)
Y102E  ; 進料手臂_(DI47)
Y102F  ; 進料手臂_(DI48)
Y1030  ; 進料手臂_(DI49)
Y1031  ; 進料手臂_(DI50)
Y1032  ; 進料手臂_(DI51)
Y1033  ; 進料手臂_(DI52)
Y1034  ; 進料手臂_(DI53)
Y1035  ; 進料手臂_(DI54)
Y1036  ; 進料手臂_(DI55)
Y1037  ; 進料手臂_(DI56)
Y1038  ; 進料手臂_(DI57)
Y1039  ; 進料手臂_(DI58)
Y103A  ; 進料手臂_(DI59)
Y103B  ; 進料手臂_(DI60)
Y103C  ; 進料手臂_(DI61)
Y103D  ; 進料手臂_(DI62)
Y103E  ; 進料手臂_(DI63)
Y103F  ; 進料手臂_(DI64)
Y1040  ; 進料手臂_(DI65)
Y1041  ; 進料手臂_(DI66)
Y1042  ; 進料手臂_(DI67)
Y1043  ; 進料手臂_(DI68)
Y1044  ; 進料手臂_(DI69)
Y1045  ; 進料手臂_(DI70)
Y1046  ; 進料手臂_(DI71)
Y1047  ; 進料手臂_(DI72)
Y1048  ; 進料手臂_(DI73)
Y1049  ; 進料手臂_(DI74)
Y104A  ; 進料手臂_(DI75)
Y104B  ; 進料手臂_(DI76)
Y104C  ; 進料手臂_(DI77)
Y104D  ; 進料手臂_(DI78)
Y104E  ; 進料手臂_(DI79)
Y104F  ; 進料手臂_(DI80)
Y1050  ; 進料手臂_(DI81)
Y1051  ; 進料手臂_(DI82)
Y1052  ; 進料手臂_(DI83)
Y1053  ; 進料手臂_(DI84)
Y1054  ; 進料手臂_(DI85)
Y1055  ; 進料手臂_(DI86)
Y1056  ; 進料手臂_(DI87)
Y1057  ; 進料手臂_(DI88)
Y1058  ; 進料手臂_(DI89)
Y1059  ; 進料手臂_(DI90)
Y105A  ; 進料手臂_(DI91)
Y105B  ; 進料手臂_(DI92)
Y105C  ; 進料手臂_(DI93)
Y105D  ; 進料手臂_(DI94)
Y105E  ; 進料手臂_(DI95)
Y105F  ; 進料手臂_(DI96)
Y1060  ; 進料手臂_(DI97)
Y1061  ; 進料手臂_(DI98)
Y1062  ; 進料手臂_(DI99)
Y1063  ; 進料手臂_(DI100)
Y1064  ; 進料手臂_(DI101)
Y1065  ; 進料手臂_(DI102)
Y1066  ; 進料手臂_(DI103)
Y1067  ; 進料手臂_(DI104)
Y1068  ; 進料手臂_(DI105)
Y1069  ; 進料手臂_(DI106)
Y106A  ; 進料手臂_(DI107)
Y106B  ; 進料手臂_(DI108)
Y106C  ; 進料手臂_(DI109)
Y106D  ; 進料手臂_(DI110)
Y106E  ; 進料手臂_(DI111)
Y106F  ; 進料手臂_(DI112)
Y1070  ; 進料手臂_(DI113)
Y1071  ; 進料手臂_(DI114)
Y1072  ; 進料手臂_(DI115)
Y1073  ; 進料手臂_(DI116)
Y1074  ; 進料手臂_(DI117)
Y1075  ; 進料手臂_(DI118)
Y1076  ; 進料手臂_(DI119)
Y1077  ; 進料手臂_(DI120)
Y1078  ; 進料手臂_(DI121)
Y1079  ; 進料手臂_(DI122)
Y107A  ; 進料手臂_(DI123)
Y107B  ; 進料手臂_(DI124)
Y107C  ; 進料手臂_(DI125)
Y107D  ; 進料手臂_(DI126)
Y107E  ; 進料手臂_(DI127)
Y107F  ; 進料手臂_(DI128)
Y1087  ; 出料手臂_(DI08)
Y1088  ; 出料手臂_(DI09)
Y1089  ; 出料手臂_(DI10)
Y108D  ; 出料手臂_(DI14)
Y1091  ; 出料手臂_(DI18)
Y1092  ; 出料手臂_(DI19)
Y1093  ; 出料手臂_(DI20)
Y1095  ; 出料手臂_(DI22)
Y1096  ; 出料手臂_(DI23)
Y1097  ; 出料手臂_(DI24)
Y1098  ; 出料手臂_(DI25)
Y1099  ; 出料手臂_(DI26)
Y109D  ; 出料手臂_(DI30)
Y109E  ; 出料手臂_(DI31)
Y109F  ; 出料手臂_(DI32)
Y10A0  ; 出料手臂_Y+20-GO(DI33)
Y10A1  ; 出料手臂_X+20-GO(DI34)
Y10A2  ; 出料手臂_Y-20(DI35)
Y10A3  ; 出料手臂_X-20(DI36)
Y10A4  ; 出料手臂_CCD再校正一次(DI37)
Y10A5  ; 出料手臂_校正位置IN38(DI38)
Y10A6  ; 出料手臂_原點往X軸移動-20MM(DI39
Y10A7  ; 出料手臂_原點往Y軸移動-20MM(DI40
Y10A8  ; 出料手臂_原點往T軸正轉移動2度
Y10A9  ; 出料手臂_(DI42)
Y10AA  ; 出料手臂_B放板待命位置(DI43)
Y10AB  ; 出料手臂_B放板上升位置(DI44)
Y10AC  ; 出料手臂_B放板完成位置(DI45)
Y10AD  ; 出料手臂_(DI46)
Y10AE  ; 出料手臂_(DI47)
Y10AF  ; 出料手臂_(DI48)
Y10B0  ; 出料手臂_(DI49)
Y10B1  ; 出料手臂_(DI50)
Y10B2  ; 出料手臂_(DI51)
Y10B3  ; 出料手臂_(DI52)
Y10B4  ; 出料手臂_(DI53)
Y10B5  ; 出料手臂_(DI54)
Y10B6  ; 出料手臂_(DI55)
Y10B7  ; 出料手臂_(DI56)
Y10B8  ; 出料手臂_(DI57)
Y10B9  ; 出料手臂_(DI58)
Y10BA  ; 出料手臂_(DI59)
Y10BB  ; 出料手臂_(DI60)
Y10BC  ; 出料手臂_(DI61)
Y10BD  ; 出料手臂_(DI62)
Y10BE  ; 出料手臂_(DI63)
Y10BF  ; 出料手臂_(DI64)
Y10C0  ; 出料手臂_(DI65)
Y10C1  ; 出料手臂_(DI66)
Y10C2  ; 出料手臂_(DI67)
Y10C3  ; 出料手臂_(DI68)
Y10C4  ; 出料手臂_(DI69)
Y10C5  ; 出料手臂_(DI70)
Y10C6  ; 出料手臂_(DI71)
Y10C7  ; 出料手臂_(DI72)
Y10C8  ; 出料手臂_(DI73)
Y10C9  ; 出料手臂_(DI74)
Y10CA  ; 出料手臂_(DI75)
Y10CB  ; 出料手臂_(DI76)
Y10CC  ; 出料手臂_(DI77)
Y10CD  ; 出料手臂_(DI78)
Y10CE  ; 出料手臂_(DI79)
Y10CF  ; 出料手臂_(DI80)
Y10D0  ; 出料手臂_(DI81)
Y10D1  ; 出料手臂_(DI82)
Y10D2  ; 出料手臂_(DI83)
Y10D3  ; 出料手臂_(DI84)
Y10D4  ; 出料手臂_(DI85)
Y10D5  ; 出料手臂_(DI86)
Y10D6  ; 出料手臂_(DI87)
Y10D7  ; 出料手臂_(DI88)
Y10D8  ; 出料手臂_(DI89)
Y10D9  ; 出料手臂_(DI90)
Y10DA  ; 出料手臂_(DI91)
Y10DB  ; 出料手臂_(DI92)
Y10DC  ; 出料手臂_(DI93)
Y10DD  ; 出料手臂_(DI94)
Y10DE  ; 出料手臂_(DI95)
Y10DF  ; 出料手臂_(DI96)
Y10E0  ; 出料手臂_(DI97)
Y10E1  ; 出料手臂_(DI98)
Y10E2  ; 出料手臂_(DI99)
Y10E3  ; 出料手臂_(DI100)
Y10E4  ; 出料手臂_(DI101)
Y10E5  ; 出料手臂_(DI102)
Y10E6  ; 出料手臂_(DI103)
Y10E7  ; 出料手臂_(DI104)
Y10E8  ; 出料手臂_(DI105)
Y10E9  ; 出料手臂_(DI106)
Y10EA  ; 出料手臂_(DI107)
Y10EB  ; 出料手臂_(DI108)
Y10EC  ; 出料手臂_(DI109)
Y10ED  ; 出料手臂_(DI110)
Y10EE  ; 出料手臂_(DI111)
Y10EF  ; 出料手臂_(DI112)
Y10F0  ; 出料手臂_(DI113)
Y10F1  ; 出料手臂_(DI114)
Y10F2  ; 出料手臂_(DI115)
Y10F3  ; 出料手臂_(DI116)
Y10F4  ; 出料手臂_(DI117)
Y10F5  ; 出料手臂_(DI118)
Y10F6  ; 出料手臂_(DI119)
Y10F7  ; 出料手臂_(DI120)
Y10F8  ; 出料手臂_(DI121)
Y10F9  ; 出料手臂_(DI122)
Y10FA  ; 出料手臂_(DI123)
Y10FB  ; 出料手臂_(DI124)
Y10FC  ; 出料手臂_(DI125)
Y10FD  ; 出料手臂_(DI126)
Y10FE  ; 出料手臂_(DI127)
Y10FF  ; 出料手臂_(DI128)
M7  ; 進料輸送停止SW
M14  ; 進料手臂下夾板  夾SW
M15  ; 進料手臂下夾板  放SW
M61  ; 框架回流輸送1   停止SW
M107  ; 出料輸送變頻器停止SW
M161  ; 左IR輸送1   停止SW
M163  ; 右IR輸送2   停止SW
M214  ; 進料手臂下夾板  夾燈
M215  ; 進料手臂下夾板  放燈
M401  ; 1
M402  ; 2
M403  ; 3
M404  ; 4
M512  ; 第13槽  循環風車SW
M513  ; 第14槽  循環風車SW
M514  ; 第15槽  循環風車SW
M515  ; 第16槽  循環風車SW
M516  ; 第17槽  循環風車SW
M517  ; 第18槽  循環風車SW
M518  ; 第19槽  循環風車SW
M519  ; 第20槽  循環風車SW
M550  ; 第01槽  循環風車燈
M551  ; 第02槽  循環風車燈
M552  ; 第03槽  循環風車燈
M553  ; 第04槽  循環風車燈
M554  ; 第05槽  循環風車燈
M555  ; 第06槽  循環風車燈
M556  ; 第07槽  循環風車燈
M557  ; 第08槽  循環風車燈
M558  ; 第09槽  循環風車燈
M559  ; 第10槽  循環風車燈
M560  ; 第11槽  循環風車燈
M561  ; 第12槽  循環風車燈
M562  ; 第13槽  循環風車燈
M563  ; 第14槽  循環風車燈
M564  ; 第15槽  循環風車燈
M565  ; 第16槽  循環風車燈
M566  ; 第17槽  循環風車燈
M567  ; 第18槽  循環風車燈
M568  ; 第19槽  循環風車燈
M569  ; 第20槽  循環風車燈
M580  ; 冷卻排氣左風車燈
M581  ; 冷卻排氣右風車燈
M582  ; 進料無塵風機燈
M583  ; 出料無塵風機燈
M584  ; 進料輸送排氣燈
M585  ; 出料輸送排氣燈
M586  ; 左冷卻  FFU風機 燈
M587  ; 右冷卻  FFU風機 燈
M612  ; 第13槽  電熱SW
M613  ; 第14槽  電熱SW
M614  ; 第15槽  電熱SW
M615  ; 第16槽  電熱SW
M616  ; 第17槽  電熱SW
M617  ; 第18槽  電熱SW
M618  ; 第19槽  電熱SW
M619  ; 第20槽  電熱SW
M650  ; 第01槽  電熱燈
M651  ; 第02槽  電熱燈
M652  ; 第03槽  電熱燈
M653  ; 第04槽  電熱燈
M654  ; 第05槽  電熱燈
M655  ; 第06槽  電熱燈
M656  ; 第07槽  電熱燈
M657  ; 第08槽  電熱燈
M658  ; 第09槽  電熱燈
M659  ; 第10槽  電熱燈
M660  ; 第11槽  電熱燈
M661  ; 第12槽  電熱燈
M662  ; 第13槽  電熱燈
M663  ; 第14槽  電熱燈
M664  ; 第15槽  電熱燈
M665  ; 第16槽  電熱燈
M666  ; 第17槽  電熱燈
M667  ; 第18槽  電熱燈
M668  ; 第19槽  電熱燈
M669  ; 第20槽  電熱燈
M712  ; 第13槽  IRA SW
M713  ; 第14槽  IRA SW
M714  ; 第15槽  IRA SW
M715  ; 第16槽  IRA SW
M716  ; 第17槽  IRA SW
M717  ; 第18槽  IRA SW
M718  ; 第19槽  IRA SW
M719  ; 第20槽  IRA SW
M732  ; 第13槽  IRB SW
M733  ; 第14槽  IRB SW
M734  ; 第15槽  IRB SW
M735  ; 第16槽  IRB SW
M736  ; 第17槽  IRB SW
M737  ; 第18槽  IRB SW
M738  ; 第19槽  IRB SW
M739  ; 第20槽  IRB SW
M750  ; 第01槽  IRA燈
M751  ; 第02槽  IRA燈
M752  ; 第03槽  IRA燈
M753  ; 第04槽  IRA燈
M754  ; 第05槽  IRA燈
M755  ; 第06槽  IRA燈
M756  ; 第07槽  IRA燈
M757  ; 第08槽  IRA燈
M758  ; 第09槽  IRA燈
M759  ; 第10槽  IRA燈
M760  ; 第11槽  IRA燈
M761  ; 第12槽  IRA燈
M762  ; 第13槽  IRA燈
M763  ; 第14槽  IRA燈
M764  ; 第15槽  IRA燈
M765  ; 第16槽  IRA燈
M766  ; 第17槽  IRA燈
M767  ; 第18槽  IRA燈
M768  ; 第19槽  IRA燈
M769  ; 第20槽  IRA燈
M770  ; 第01槽  IRB燈
M771  ; 第02槽  IRB燈
M772  ; 第03槽  IRB燈
M773  ; 第04槽  IRB燈
M774  ; 第05槽  IRB燈
M775  ; 第06槽  IRB燈
M776  ; 第07槽  IRB燈
M777  ; 第08槽  IRB燈
M778  ; 第09槽  IRB燈
M779  ; 第10槽  IRB燈
M780  ; 第11槽  IRB燈
M781  ; 第12槽  IRB燈
M782  ; 第13槽  IRB燈
M783  ; 第14槽  IRB燈
M784  ; 第15槽  IRB燈
M785  ; 第16槽  IRB燈
M786  ; 第17槽  IRB燈
M787  ; 第18槽  IRB燈
M788  ; 第19槽  IRB燈
M789  ; 第20槽  IRB燈
M1002  ; 進料牙叉機構回原點SW
M1012  ; 出料牙叉機構回原點SW
M1013  ; 出料手臂機構回原點SW
M1052  ; 進料牙叉機構回原點燈
M1062  ; 出料牙叉機構回原點燈
M1063  ; 出料手臂機構回原點燈
M1123  ; 進料整板位置04 SW
M1124  ; 進料整板位置05 SW
M1125  ; 進料整板位置06 SW
M1126  ; 進料整板位置07 SW
M1127  ; 進料整板位置08 SW
M1128  ; 進料整板位置09 SW
M1129  ; 進料整板位置10 SW
M1143  ; 進料整板位置04燈
M1144  ; 進料整板位置05燈
M1145  ; 進料整板位置06燈
M1146  ; 進料整板位置07燈
M1147  ; 進料整板位置08燈
M1148  ; 進料整板位置09燈
M1149  ; 進料整板位置10燈
M1222  ; 牙插移載位置03 SW
M1223  ; 牙插移載位置04 SW
M1224  ; 牙插移載位置05 SW
M1225  ; 牙插移載位置06 SW
M1226  ; 牙插移載位置07 SW
M1227  ; 牙插移載位置08 SW
M1228  ; 牙插移載位置09 SW
M1229  ; 牙插移載位置10 SW
M1242  ; 牙插移載位置03燈
M1243  ; 牙插移載位置04燈
M1244  ; 牙插移載位置05燈
M1245  ; 牙插移載位置06燈
M1246  ; 牙插移載位置07燈
M1247  ; 牙插移載位置08燈
M1248  ; 牙插移載位置09燈
M1249  ; 牙插移載位置10燈
M1422  ; 進手臂取手位置03 SW
M1423  ; 進手臂取手位置04 SW
M1424  ; 進手臂取手位置05 SW
M1425  ; 進手臂取手位置06 SW
M1426  ; 進手臂取手位置07 SW
M1427  ; 進手臂取手位置08 SW
M1428  ; 進手臂取手位置09 SW
M1429  ; 進手臂取手位置10 SW
M1442  ; 進手臂取手位置03燈
M1443  ; 進手臂取手位置04燈
M1444  ; 進手臂取手位置05燈
M1445  ; 進手臂取手位置06燈
M1446  ; 進手臂取手位置07燈
M1447  ; 進手臂取手位置08燈
M1448  ; 進手臂取手位置09燈
M1449  ; 進手臂取手位置10燈
M1524  ; 進料托框昇降位置05 SW
M1525  ; 進料托框昇降位置06 SW
M1526  ; 進料托框昇降位置07 SW
M1527  ; 進料托框昇降位置08 SW
M1528  ; 進料托框昇降位置09 SW
M1529  ; 進料托框昇降位置10 SW
M1544  ; 進料托框昇降位置05燈
M1545  ; 進料托框昇降位置06燈
M1546  ; 進料托框昇降位置07燈
M1547  ; 進料托框昇降位置08燈
M1548  ; 進料托框昇降位置09燈
M1549  ; 進料托框昇降位置10燈
M1550  ; 進料托框昇降位置01 SW*
M1551  ; 進料托框昇降位置02 SW*
M1552  ; 進料托框昇降位置03 SW*
M1553  ; 進料托框昇降位置04 SW*
M1554  ; 進料托框昇降位置05 SW*
M1555  ; 進料托框昇降位置06 SW*
M1556  ; 進料托框昇降位置07 SW*
M1557  ; 進料托框昇降位置08 SW*
M1558  ; 進料托框昇降位置09 SW*
M1559  ; 進料托框昇降位置10 SW*
M1625  ; 進左開爪位置06 SW
M1626  ; 進左開爪位置07 SW
M1627  ; 進左開爪位置08 SW
M1628  ; 進左開爪位置09 SW
M1629  ; 進左開爪位置10 SW
M1645  ; 進左開爪位置06燈
M1646  ; 進左開爪位置07燈
M1647  ; 進左開爪位置08燈
M1648  ; 進左開爪位置09燈
M1649  ; 進左開爪位置10燈
M1725  ; 進右開爪位置06 SW
M1726  ; 進右開爪位置07 SW
M1727  ; 進右開爪位置08 SW
M1728  ; 進右開爪位置09 SW
M1729  ; 進右開爪位置10 SW
M1745  ; 進右開爪位置06燈
M1746  ; 進右開爪位置07燈
M1747  ; 進右開爪位置08燈
M1749  ; 進右開爪位置10燈
M1829  ; CCD_HeartBeat心跳
M1857  ; 進料牙叉上昇位置
M1858  ; 進料牙叉下降位置
M1860  ; CCD 對位逾時計次到達
M1873  ; CCD 重置PB
M1875  ; 品種切換PB
M1881  ; CCD基準位置登錄燈
M1883  ; CCD重置燈
M1884  ; Y+20
M1885  ; X-20
M1886  ; Y-20
M1890  ; CCD 重置PLS
M1891  ; 搜索OK  完成
M1892  ; 發生搜索錯誤
M1895  ; 搜索結束PLS
M1897  ; 出料主傳動有板燈
M2123  ; 分流前取框位置04 SW
M2124  ; 分流前取框位置05 SW
M2125  ; 分流前取框位置06 SW
M2126  ; 分流前取框位置07 SW
M2127  ; 分流前取框位置08 SW
M2128  ; 分流前取框位置09 SW
M2129  ; 分流前取框位置10 SW
M2143  ; 分流前取框位置04燈
M2144  ; 分流前取框位置05燈
M2145  ; 分流前取框位置06燈
M2146  ; 分流前取框位置07燈
M2147  ; 分流前取框位置08燈
M2148  ; 分流前取框位置09燈
M2149  ; 分流前取框位置10燈
M2223  ; 合流後掛框位置04 SW
M2224  ; 合流後掛框位置05 SW
M2225  ; 合流後掛框位置06 SW
M2226  ; 合流後掛框位置07 SW
M2227  ; 合流後掛框位置08 SW
M2228  ; 合流後掛框位置09 SW
M2229  ; 合流後掛框位置10 SW
M2243  ; 合流後掛框位置04燈
M2244  ; 合流後掛框位置05燈
M2245  ; 合流後掛框位置06燈
M2246  ; 合流後掛框位置07燈
M2247  ; 合流後掛框位置08燈
M2248  ; 合流後掛框位置09燈
M2249  ; 合流後掛框位置10燈
M2256  ; 出料平台位置07 SW*
M2257  ; 出料平台位置08 SW*
M2258  ; 出料平台位置09 SW*
M2259  ; 出料平台位置10 SW*
M3123  ; 出手臂取手位置04 SW
M3124  ; 出手臂取手位置05 SW
M3125  ; 出手臂取手位置06 SW
M3126  ; 出手臂取手位置07 SW
M3127  ; 出手臂取手位置08 SW
M3128  ; 出手臂取手位置09 SW
M3129  ; 出手臂取手位置10 SW
M3143  ; 出手臂取手位置04燈
M3144  ; 出手臂取手位置05燈
M3145  ; 出手臂取手位置06燈
M3146  ; 出手臂取手位置07燈
M3147  ; 出手臂取手位置08燈
M3148  ; 出手臂取手位置09燈
M3149  ; 出手臂取手位置10燈
M3225  ; 出料托框昇降位置06 SW
M3226  ; 出料托框昇降位置07 SW
M3227  ; 出料托框昇降位置08 SW
M3228  ; 出料托框昇降位置09 SW
M3229  ; 出料托框昇降位置10 SW
M3245  ; 出料托框昇降位置06燈
M3246  ; 出料托框昇降位置07燈
M3247  ; 出料托框昇降位置08燈
M3248  ; 出料托框昇降位置09燈
M3249  ; 出料托框昇降位置10燈
M3325  ; 出左開夾位置06 SW
M3326  ; 出左開夾位置07 SW
M3327  ; 出左開夾位置08 SW
M3328  ; 出左開夾位置09 SW
M3329  ; 出左開夾位置10 SW
M3345  ; 出左開夾位置06燈
M3346  ; 出左開夾位置07燈
M3347  ; 出左開夾位置08燈
M3348  ; 出左開夾位置09燈
M3349  ; 出左開夾位置10燈
M3353  ; 旋轉位置04 SW*
M3354  ; 旋轉位置05 SW*
M3355  ; 旋轉位置06 SW*
M3356  ; 旋轉位置07 SW*
M3357  ; 旋轉位置08 SW*
M3358  ; 旋轉位置09 SW*
M3359  ; 旋轉位置10 SW*
M3425  ; 出右開夾位置06 SW
M3426  ; 出右開夾位置07 SW
M3427  ; 出右開夾位置08 SW
M3428  ; 出右開夾位置09 SW
M3429  ; 出右開夾位置10 SW
M3445  ; 出右開夾位置06燈
M3446  ; 出右開夾位置07燈
M3447  ; 出右開夾位置08燈
M3448  ; 出右開夾位置09燈
M3449  ; 出右開夾位置10燈
M3523  ; 出板牙插移載位置04 SW
M3524  ; 出板牙插移載位置05 SW
M3525  ; 出板牙插移載位置06 SW
M3526  ; 出板牙插移載位置07 SW
M3527  ; 出板牙插移載位置08 SW
M3528  ; 出板牙插移載位置09 SW
M3529  ; 出板牙插移載位置10 SW
M3543  ; 出板牙插移載位置04燈
M3544  ; 出板牙插移載位置05燈
M3545  ; 出板牙插移載位置06燈
M3546  ; 出板牙插移載位置07燈
M3547  ; 出板牙插移載位置08燈
M3548  ; 出板牙插移載位置09燈
M3549  ; 出板牙插移載位置10燈
M4058  ; 預留正極限異常
M4059  ; 預留負極限異常
M4070  ; 預留正極限異常
M4071  ; 預留負極限異常
M4149  ; 進料輸送減速光電異常
M4209  ; 合流右_旋轉定點異常
M4301  ; 第02槽   OTP超溫
M4302  ; 第03槽   OTP超溫
M4303  ; 第04槽   OTP超溫
M4304  ; 第05槽   OTP超溫
M4305  ; 第06槽   OTP超溫
M4306  ; 第07槽   OTP超溫
M4307  ; 第08槽   OTP超溫
M4321  ; 第02槽  IRA OTP 超溫
M4322  ; 第03槽  IRA OTP 超溫
M4323  ; 第04槽  IRA OTP 超溫
M4324  ; 第05槽  IRA OTP 超溫
M4325  ; 第06槽  IRA OTP 超溫
M4326  ; 第07槽  IRA OTP 超溫
M4327  ; 第08槽  IRA OTP 超溫
M4341  ; 第02槽  IRB OTP 超溫
M4342  ; 第03槽  IRB OTP 超溫
M4343  ; 第04槽  IRB OTP 超溫
M4344  ; 第05槽  IRB OTP 超溫
M4345  ; 第06槽  IRB OTP 超溫
M4346  ; 第07槽  IRB OTP 超溫
M4351  ; 第12槽  IRB OTP 超溫
M4421  ; 第02槽 熱風低溫異常
M4422  ; 第03槽 熱風低溫異常
M4423  ; 第04槽 熱風低溫異常
M4424  ; 第05槽 熱風低溫異常
M4425  ; 第06槽 熱風低溫異常
M4426  ; 第07槽 熱風低溫異常
M4427  ; 第08槽 熱風低溫異常
M4428  ; 第09槽 熱風低溫異常
M4429  ; 第10槽 熱風低溫異常
M4430  ; 第11槽 熱風低溫異常
M4431  ; 第12槽 熱風低溫異常
M4441  ; 第02槽 IRA 低溫異常
M4442  ; 第03槽 IRA 低溫異常
M4443  ; 第04槽 IRA 低溫異常
M4444  ; 第05槽 IRA 低溫異常
M4445  ; 第06槽 IRA 低溫異常
M4446  ; 第07槽 IRA 低溫異常
M4447  ; 第08槽 IRA 低溫異常
M4448  ; 第09槽 IRA 低溫異常
M4449  ; 第10槽 IRA 低溫異常
M4450  ; 第11槽 IRA 低溫異常
M4451  ; 第12槽 IRA 低溫異常
M4461  ; 第02槽 IRB 低溫異常
M4462  ; 第03槽 IRB 低溫異常
M4463  ; 第04槽 IRB 低溫異常
M4464  ; 第05槽 IRB 低溫異常
M4465  ; 第06槽 IRB 低溫異常
M4466  ; 第07槽 IRB 低溫異常
M4467  ; 第08槽 IRB 低溫異常
M4468  ; 第09槽 IRB 低溫異常
M4469  ; 第10槽 IRB 低溫異常
M4470  ; 第11槽 IRB 低溫異常
M4471  ; 第12槽 IRB 低溫異常
M4481  ; 第02槽 熱風超溫異常
M4482  ; 第03槽 熱風超溫異常
M4483  ; 第04槽 熱風超溫異常
M4484  ; 第05槽 熱風超溫異常
M4485  ; 第06槽 熱風超溫異常
M4486  ; 第07槽 熱風超溫異常
M4487  ; 第08槽 熱風超溫異常
M4501  ; 第2槽 IRA 超溫異常
M4502  ; 第3槽 IRA 超溫異常
M4503  ; 第4槽 IRA 超溫異常
M4504  ; 第5槽 IRA 超溫異常
M4505  ; 第6槽 IRA 超溫異常
M4506  ; 第7槽 IRA 超溫異常
M4507  ; 第8槽 IRA 超溫異常
M4512  ; 第13槽 IRA 超溫異常
M4513  ; 第14槽 IRA 超溫異常
M4514  ; 第15槽 IRA 超溫異常
M4515  ; 第16槽 IRA 超溫異常
M4521  ; 第2槽 IRB 超溫異常
M4522  ; 第3槽 IRB 超溫異常
M4523  ; 第4槽 IRB 超溫異常
M4524  ; 第5槽 IRB 超溫異常
M4525  ; 第6槽 IRB 超溫異常
M4526  ; 第7槽 IRB 超溫異常
M4527  ; 第8槽 IRB 超溫異常
M4532  ; 第13槽 IRB 超溫異常
M4533  ; 第14槽 IRB 超溫異常
M4534  ; 第15槽 IRB 超溫異常
M4535  ; 第16槽 IRB 超溫異常
M4621  ; 取板牙插驅動器電池異常
M4623  ; 進料手臂取手驅動器電池異常
M4624  ; 進料托框昇降驅動器電池異常
M4625  ; 進左開夾驅動器電池異常
M4626  ; 進右開夾驅動器電池異常
M4630  ; 出料手臂取手驅動器電池異常
M4631  ; 出料托框昇降驅動器電池異常
M4632  ; 出左開夾驅動器電池異常
M4633  ; 出右開夾驅動器電池異常
M4681  ; 取板牙插歸零要求異常
M4683  ; 進料手臂取手歸零要求異常
M4684  ; 進料托框昇降歸零要求異常
M4685  ; 進左開夾歸零要求異常
M4686  ; 進右開夾歸零要求異常
M4687  ; 分流前取框歸零要求異常
M4688  ; 出板牙插歸零要求異常
M4690  ; 出料手臂取手歸零要求異常
M4691  ; 出料托框昇降歸零要求異常
M4692  ; 出左開夾歸零要求異常
M4693  ; 出右開夾歸零要求異常
M4694  ; 合流後掛框歸零要求異常
M4744  ; 印刷機左圍籬安全門偵測ˋ異常
M4745  ; 印刷機右圍籬安全門偵測ˋ異常
M4920  ; 入口計數自保持
M4934  ; 上位允許放板START
M4943  ; 上位下GO_REMOTE
M4944  ; 上位下GO-LOCAL
M5130  ; 回上位面板#1入板訊號
M5135  ; 回上位Panel#1出板訊號
M5150  ; 進料板材尺寸連線模式燈
M5151  ; 出料板材尺寸連線模式燈
M5200  ; 進料I/O測試
M5201  ; 進料I/O 測試_01
M5202  ; 進料I/O 測試_02
M5203  ; 進料I/O 測試_03
M5204  ; 進料I/O 測試_04
M5205  ; 進料I/O 測試_05
M5206  ; 進料I/O 測試_06
M5207  ; 進料I/O 測試_07
M5208  ; 進料I/O 測試_08
M5209  ; 進料I/O 測試_09
M5210  ; 進料I/O 測試_10
M5211  ; 進料I/O 測試_11
M5212  ; 進料I/O 測試_12
M5213  ; 進料I/O 測試_13
M5214  ; 進料I/O 測試_14
M5215  ; 進料I/O 測試_15
M5216  ; 進料I/O 測試_16
M5220  ; 出料I/O測試
M5221  ; 出料I/O 測試_01
M5222  ; 出料I/O 測試_02
M5223  ; 出料I/O 測試_03
M5224  ; 出料I/O 測試_04
M5225  ; 出料I/O 測試_05
M5226  ; 出料I/O 測試_06
M5227  ; 出料I/O 測試_07
M5228  ; 出料I/O 測試_08
M5229  ; 出料I/O 測試_09
M5230  ; 出料I/O 測試_10
M5231  ; 出料I/O 測試_11
M5232  ; 出料I/O 測試_12
M5233  ; 出料I/O 測試_13
M5234  ; 出料I/O 測試_14
M5235  ; 出料I/O 測試_15
M5236  ; 出料I/O 測試_16
M5320  ; FX機台狀態改變
M5410  ; 出料手臂至校正位置手動
M5422  ; 出料手臂自動取板等待點動作條件
M5502  ; PC->Start command
M5503  ; PC->Stop command
M5507  ; 進料開爪位置有板BF
M5508  ; 進料入爐有板BF
M5510  ; 機台狀態BF
M5511  ; 機台狀態INIT
M5512  ; 機台狀態Idle
M5513  ; 機台狀態Ready
M5514  ; 機台狀態Warmup
M5515  ; 機台狀態Exccuting
M5516  ; 機台狀態Pause
M5517  ; 機台狀態Maintenance
M5520  ; 進料段ALARM
M5521  ; 進料段有料
M5522  ; 進料段MOVING
M5523  ; 爐體段ALARM
M5524  ; 爐體段有料
M5525  ; 出料段ALARM
M5526  ; 出料段有料
M5527  ; 出料段MOVING
M5528  ; 回流段ALARM
M5530  ; 機台內有板
M5532  ; 機台LOT生產完畢KP
M6059  ; Host刪除配方
M6060  ; Host刪除配方完成
M6105  ; 回上位新增配方
M6106  ; 回上位刪除配方
M6134  ; 三色燈狀態改變
M6137  ; 手動
M6140  ; 要求上位回讀工單板號右爐
M6141  ; 要求上位回讀工單右爐
M6142  ; 三色黃燈
M6218  ; 和上位連線中
M7017  ; 配方切換旗標
M7022  ; 配方搜尋比對OK
M7026  ; 去空白KP
M7030  ; 配方寫入-KP
M7031  ; 配方寫入-KP
M7035  ; 配方空白
M7040  ; 入口計數自保持
M7042  ; 回上位面板#1入板訊號
M7043  ; 回上位Panel#1出板訊號
M7075  ; 批數歸零旗標
M7076  ; 爐內片數歸零PB
M7077  ; 批次數量歸零PB
M7084  ; TEST
M7120  ; 比對GO-REMOTE字串不對
M7121  ; 名稱GO-LOCAL比對不對
M7122  ; 比對RESUME字串不對
M7123  ; 比對PPID字串不對
M7124  ; 比對PAUSE字串不對
M7125  ; 比對START字串不對
M7126  ; 比對STOP字串不對
M7127  ; 比對PP_SELECT字串不對
M7142  ; [HH-02] 配方搜尋比對NG
M7170  ; [PPID]  配方搜尋比對OK_配方可
M7203  ; 未知?測試用
M7207  ; 上位切換成GO-REMOTE
M7208  ; 上位切換成GO-LOCAL
M7214  ; SECS上位下指令觸發Cmd-燈號
M7322  ; 程式結束
M7604  ; ALARM   暫停
M7605  ; 進料回流光纖暫停
L14  ; 允許進料手臂下夾板  夾
L15  ; 允許進料手臂下夾板  放
L100  ; 停電保持SECS    手動/自動連線
L201  ; Disable Check   FrameL/D
L202  ; Disable Check   SEN. L/D
L203  ; Disable Check   FrameU/D
L204  ; Disable Check   SEN. U/D
L205  ; Disable Check   FrameR/F
L206  ; Disable Check   SEN. R/F
L226  ; 進料牙叉吸風使用
L251  ; 夾爪彈簧偵測
L512  ; 第13槽  循環風車SW  PLS
L513  ; 第14槽  循環風車SW  PLS
L514  ; 第15槽  循環風車SW  PLS
L515  ; 第16槽  循環風車SW  PLS
L516  ; 第17槽  循環風車SW  PLS
L517  ; 第18槽  循環風車SW  PLS
L518  ; 第19槽  循環風車SW  PLS
L519  ; 第20槽  循環風車SW  PLS
L552  ; 第13槽  電熱SW  PLS
L553  ; 第14槽  電熱SW  PLS
L554  ; 第15槽  電熱SW  PLS
L555  ; 第16槽  電熱SW  PLS
L556  ; 第17槽  電熱SW  PLS
L557  ; 第18槽  電熱SW  PLS
L558  ; 第19槽  電熱SW  PLS
L559  ; 第20槽  電熱SW  PLS
L572  ; 第13槽  IRA SW  PLS
L573  ; 第14槽  IRA SW  PLS
L574  ; 第15槽  IRA SW  PLS
L575  ; 第16槽  IRA SW  PLS
L576  ; 第17槽  IRA SW  PLS
L577  ; 第18槽  IRA SW  PLS
L578  ; 第19槽  IRA SW  PLS
L579  ; 第20槽  IRA SW  PLS
L592  ; 第13槽  IRB SW  PLS
L593  ; 第14槽  IRB SW  PLS
L594  ; 第15槽  IRB SW  PLS
L595  ; 第16槽  IRB SW  PLS
L596  ; 第17槽  IRB SW  PLS
L597  ; 第18槽  IRB SW  PLS
L598  ; 第19槽  IRB SW  PLS
L599  ; 第20槽  IRB SW  PLS
L612  ; 第13槽  循環風車
L613  ; 第14槽  循環風車
L614  ; 第15槽  循環風車
L615  ; 第16槽  循環風車
L616  ; 第17槽  循環風車
L617  ; 第18槽  循環風車
L618  ; 第19槽  循環風車
L619  ; 第20槽  循環風車
L652  ; 第13槽  電熱
L653  ; 第14槽  電熱
L654  ; 第15槽  電熱
L655  ; 第16槽  電熱
L656  ; 第17槽  電熱
L657  ; 第18槽  電熱
L658  ; 第19槽  電熱
L659  ; 第20槽  電熱
L672  ; 第13槽  IRA
L673  ; 第14槽  IRA
L674  ; 第15槽  IRA
L675  ; 第16槽  IRA
L676  ; 第17槽  IRA
L677  ; 第18槽  IRA
L678  ; 第19槽  IRA
L679  ; 第20槽  IRA
L692  ; 第13槽  IRB
L693  ; 第14槽  IRB
L694  ; 第15槽  IRB
L695  ; 第16槽  IRB
L696  ; 第17槽  IRB
L697  ; 第18槽  IRB
L698  ; 第19槽  IRB
L699  ; 第20槽  IRB
L700  ; 低溫異常01
L701  ; 低溫異常02
L702  ; 低溫異常03
L703  ; 低溫異常04
L704  ; 低溫異常05
L705  ; 低溫異常06
L706  ; 低溫異常07
L707  ; 低溫異常08
L708  ; 低溫異常09
L709  ; 低溫異常10
L710  ; 低溫異常11
L711  ; 低溫異常12
L1030  ; 步進計時到PLS
L1031  ; 倒數允許進料
L1032  ; 倒數允許出料
L1103  ; 整板  STOP
L1111  ; 速度轉換位置
L1118  ; 整板伺服啟動
L1119  ; 整板伺服啟動異常
L1129  ; 整板己回原點
L1134  ; 進料整板位置05
L1135  ; 進料整板位置06
L1136  ; 進料整板位置07
L1137  ; 進料整板位置08
L1138  ; 進料整板位置09
L1139  ; 進料整板位置10
L1144  ; 整板位置05 訊號
L1145  ; 整板位置06 訊號
L1146  ; 整板位置07 訊號
L1147  ; 整板位置08 訊號
L1148  ; 整板位置09 訊號
L1171  ; 整板速度轉換位置
L1172  ; 整板命令近點
L1173  ; 整板歸零要求
L1174  ; 整板歸零完成
L1185  ; 整板Positioning complete
L1203  ; 牙插移載  STOP
L1211  ; 牙插移載速度轉換位置
L1218  ; 牙插移載伺服啟動
L1219  ; 牙插移載伺服啟動異常
L1229  ; 牙插移載己回原點
L1239  ; 牙插移載位置10
L1244  ; 牙插移載位置05 訊號
L1245  ; 牙插移載位置06 訊號
L1246  ; 牙插移載位置07 訊號
L1247  ; 牙插移載位置08 訊號
L1248  ; 牙插移載位置09 訊號
L1249  ; 牙插移載位置10 訊號
L1271  ; 牙插移載速度轉換位置
L1272  ; 牙插移載命令近點
L1273  ; 牙插移載歸零要求
L1274  ; 牙插移載歸零完成
L1285  ; 移載Positioning complete
L1403  ; 進手臂取手STOP
L1411  ; 進手臂取手速度轉換位置
L1418  ; 進手臂取手伺服啟動
L1419  ; 進手臂取手伺服啟動異常
L1429  ; 進手臂取手己回原點
L1439  ; 進手臂取手位置10
L1444  ; 進手臂取手位置05 訊號
L1445  ; 進手臂取手位置06 訊號
L1446  ; 進手臂取手位置07 訊號
L1447  ; 進手臂取手位置08 訊號
L1448  ; 進手臂取手位置09 訊號
L1449  ; 進手臂取手位置10 訊號
L1471  ; 進手臂取手速度轉換位置
L1472  ; 進手臂取手命令近點
L1473  ; 進手臂取手歸零要求
L1474  ; 進手臂取手歸零完成
L1485  ; 進手臂取手Positioning complete
L1503  ; 進料托框昇降STOP
L1511  ; 進料托框昇降速度轉換位置
L1518  ; 進料托框昇降伺服啟動
L1519  ; 進料托框昇降伺服啟動異常
L1529  ; 進料托框昇降己回原點
L1545  ; 進料托框昇降位置06 訊號
L1546  ; 進料托框昇降位置07 訊號
L1547  ; 進料托框昇降位置08 訊號
L1548  ; 進料托框昇降位置09 訊號
L1549  ; 進料托框昇降位置10 訊號
L1571  ; 進料托框昇降速度轉換位置
L1572  ; 進料托框昇降命令近點
L1573  ; 進料托框昇降歸零要求
L1574  ; 進料托框昇降歸零完成
L1585  ; 進料托框昇降Positioning complete
L1603  ; 進左開爪STOP
L1611  ; 進左開爪速度轉換位置
L1618  ; 進左開爪伺服啟動
L1619  ; 進左開爪伺服啟動異常
L1629  ; 進左開爪己回原點
L1639  ; 進左開爪位置10
L1645  ; 進左開爪位置06 訊號
L1646  ; 進左開爪位置07 訊號
L1647  ; 進左開爪位置08 訊號
L1648  ; 進左開爪位置09 訊號
L1649  ; 進左開爪位置10 訊號
L1671  ; 進左開爪速度轉換位置
L1672  ; 進左開爪命令近點
L1673  ; 進左開爪歸零要求
L1674  ; 進左開爪歸零完成
L1685  ; 進左開爪Positioning complete
L1703  ; 進右開爪STOP
L1711  ; 進右開爪速度轉換位置
L1718  ; 進右開爪伺服啟動
L1719  ; 進右開爪伺服啟動異常
L1729  ; 進右開爪己回原點
L1739  ; 進右開爪位置10
L1745  ; 進右開爪位置06 訊號
L1746  ; 進右開爪位置07 訊號
L1747  ; 進右開爪位置08 訊號
L1748  ; 進右開爪位置09 訊號
L1749  ; 進右開爪位置10 訊號
L1771  ; 進右開爪速度轉換位置
L1772  ; 進右開爪命令近點
L1773  ; 進右開爪歸零要求
L1774  ; 進右開爪歸零完成
L1785  ; 進右開爪Positioning complete
L1800  ; 進料左側框架退出
L1810  ; 進料右側框架退出
L1820  ; 出料左側框架退出
L1830  ; 出料右側框架退出
L2103  ; 分流前取框STOP
L2111  ; 分流前取框速度轉換位置
L2118  ; 分流前取框伺服啟動
L2119  ; 分流前取框伺服啟動異常
L2129  ; 分流前取框己回原點
L2139  ; 分流前取框位置10
L2144  ; 分流前取框位置05 訊號
L2145  ; 分流前取框位置06 訊號
L2146  ; 分流前取框位置07 訊號
L2147  ; 分流前取框位置08 訊號
L2148  ; 分流前取框位置09 訊號
L2149  ; 分流前取框位置10 訊號
L2171  ; 分流前取框速度轉換位置
L2172  ; 分流前取框命令近點
L2173  ; 分流前取框歸零要求
L2174  ; 分流前取框歸零完成
L2185  ; 分流前取框Positioning complete
L2203  ; 合流後掛框STOP
L2211  ; 合流後掛框速度轉換位置
L2218  ; 合流後掛框伺服啟動
L2219  ; 合流後掛框伺服啟動異常
L2229  ; 合流後掛框己回原點
L2239  ; 合流後掛框位置10
L2244  ; 合流後掛框位置05 訊號
L2245  ; 合流後掛框位置06 訊號
L2246  ; 合流後掛框位置07 訊號
L2247  ; 合流後掛框位置08 訊號
L2248  ; 合流後掛框位置09 訊號
L2249  ; 合流後掛框位置10 訊號
L2271  ; 合流後掛框速度轉換位置
L2272  ; 合流後掛框命令近點
L2273  ; 合流後掛框歸零要求
L2274  ; 合流後掛框歸零完成
L2285  ; 合流後掛框Positioning complete
L2292  ; 允許合流取框位置03
L2808  ; 第09站  CC-LINK 異常
L2809  ; 第10站  CC-LINK 異常
L2810  ; 第11站  CC-LINK 異常
L2811  ; 第12站  CC-LINK 異常
L2812  ; 第13站  CC-LINK 異常
L2813  ; 第14站  CC-LINK 異常
L2814  ; 第15站  CC-LINK 異常
L2815  ; 第16站  CC-LINK 異常
L2816  ; 第17站  CC-LINK 異常
L2817  ; 第18站  CC-LINK 異常
L2818  ; 第19站  CC-LINK 異常
L2819  ; 第20站  CC-LINK 異常
L2820  ; 第21站  CC-LINK 異常
L2821  ; 第22站  CC-LINK 異常
L2822  ; 第23站  CC-LINK 異常
L2823  ; 第24站  CC-LINK 異常
L2824  ; 第25站  CC-LINK 異常
L2825  ; 第26站  CC-LINK 異常
L2826  ; 第27站  CC-LINK 異常
L2827  ; 第28站  CC-LINK 異常
L2828  ; 第29站  CC-LINK 異常
L2829  ; 第30站  CC-LINK 異常
L2830  ; 第31站  CC-LINK 異常
L2831  ; 第32站  CC-LINK 異常
L2832  ; 第33站  CC-LINK 異常
L2833  ; 第34站  CC-LINK 異常
L2834  ; 第35站  CC-LINK 異常
L2835  ; 第36站  CC-LINK 異常
L2836  ; 第37站  CC-LINK 異常
L2837  ; 第38站  CC-LINK 異常
L2838  ; 第39站  CC-LINK 異常
L2839  ; 第40站  CC-LINK 異常
L2840  ; 第41站  CC-LINK 異常
L2841  ; 第42站  CC-LINK 異常
L2842  ; 第43站  CC-LINK 異常
L2843  ; 第44站  CC-LINK 異常
L2844  ; 第45站  CC-LINK 異常
L2845  ; 第46站  CC-LINK 異常
L2846  ; 第47站  CC-LINK 異常
L2847  ; 第48站  CC-LINK 異常
L2848  ; 第49站  CC-LINK 異常
L2849  ; 第50站  CC-LINK 異常
L2850  ; 第51站  CC-LINK 異常
L2851  ; 第52站  CC-LINK 異常
L2852  ; 第53站  CC-LINK 異常
L2853  ; 第54站  CC-LINK 異常
L2854  ; 第55站  CC-LINK 異常
L2855  ; 第56站  CC-LINK 異常
L2856  ; 第57站  CC-LINK 異常
L2857  ; 第58站  CC-LINK 異常
L2858  ; 第59站  CC-LINK 異常
L2859  ; 第60站  CC-LINK 異常
L2860  ; 第61站  CC-LINK 異常
L2861  ; 第62站  CC-LINK 異常
L2862  ; 第63站  CC-LINK 異常
L2863  ; 第64站  CC-LINK 異常
L2872  ; Unload_ CC-Link OK
L3103  ; 出手臂取手STOP
L3111  ; 出手臂取手速度轉換位置
L3118  ; 出手臂取手伺服啟動
L3119  ; 出手臂取手伺服啟動異常
L3129  ; 出手臂取手己回原點
L3139  ; 出手臂取手位置10
L3144  ; 出手臂取手位置05 訊號
L3145  ; 出手臂取手位置06 訊號
L3146  ; 出手臂取手位置07 訊號
L3147  ; 出手臂取手位置08 訊號
L3148  ; 出手臂取手位置09 訊號
L3149  ; 出手臂取手位置10 訊號
L3171  ; 出手臂取手速度轉換位置
L3172  ; 出手臂取手命令近點
L3173  ; 出手臂取手歸零要求
L3174  ; 出手臂取手歸零完成
L3185  ; 出手臂取手Positioning complete
L3190  ; 出料手臂移載允許位置01  訊號*
L3203  ; 出料托框昇降STOP
L3211  ; 出料托框昇降速度轉換位置
L3218  ; 出料托框昇降伺服啟動
L3219  ; 出料托框昇降伺服啟動異常
L3229  ; 出料托框昇降己回原點
L3245  ; 出料托框昇降位置06 訊號
L3246  ; 出料托框昇降位置07 訊號
L3247  ; 出料托框昇降位置08 訊號
L3248  ; 出料托框昇降位置09 訊號
L3249  ; 出料托框昇降位置10 訊號
L3271  ; 出料托框昇降速度轉換位置
L3272  ; 出料托框昇降命令近點
L3273  ; 出料托框昇降歸零要求
L3274  ; 出料托框昇降歸零完成
L3285  ; 出料托框昇降Positioning complete
L3290  ; 出料手臂昇降允許位置01  訊號*
L3303  ; 出左開夾STOP
L3311  ; 出左開夾速度轉換位置
L3318  ; 出左開夾伺服啟動
L3319  ; 出左開夾伺服啟動異常
L3329  ; 出左開夾己回原點
L3339  ; 出左開夾位置10
L3345  ; 出左開夾位置06 訊號
L3346  ; 出左開夾位置07 訊號
L3347  ; 出左開夾位置08 訊號
L3348  ; 出左開夾位置09 訊號
L3349  ; 出左開夾位置10 訊號
L3371  ; 出左開夾速度轉換位置
L3372  ; 出左開夾命令近點
L3373  ; 出左開夾歸零要求
L3374  ; 出左開夾歸零完成
L3385  ; 出左開夾Positioning complete
L3403  ; 出右開夾STOP
L3411  ; 出右開夾速度轉換位置
L3418  ; 出右開夾伺服啟動
L3419  ; 出右開夾伺服啟動異常
L3429  ; 出右開夾己回原點
L3439  ; 出右開夾位置10
L3445  ; 出右開夾位置06 訊號
L3446  ; 出右開夾位置07 訊號
L3447  ; 出右開夾位置08 訊號
L3448  ; 出右開夾位置09 訊號
L3449  ; 出右開夾位置10 訊號
L3471  ; 出右開夾速度轉換位置
L3472  ; 出右開夾命令近點
L3473  ; 出右開夾歸零要求
L3474  ; 出右開夾歸零完成
L3485  ; 出右開夾Positioning complete
L3503  ; 出板牙插移載STOP
L3511  ; 出板牙插移載速度轉換位置
L3518  ; 出板牙插移載伺服啟動
L3519  ; 出板牙插移載伺服啟動異常
L3529  ; 出板牙插移載己回原點
L3539  ; 出板牙插移載位置10
L3544  ; 出板牙插移載位置05 訊號
L3545  ; 出板牙插移載位置06 訊號
L3546  ; 出板牙插移載位置07 訊號
L3547  ; 出板牙插移載位置08 訊號
L3548  ; 出板牙插移載位置09 訊號
L3549  ; 出板牙插移載位置10 訊號
L3571  ; 出板牙插移載速度轉換位置
L3572  ; 出板牙插移載命令近點
L3573  ; 出板牙插移載歸零要求
L3574  ; 出板牙插移載歸零完成
L3585  ; 出板牙插移載Positioning complete
L3652  ; 下料手動允許信號
L3662  ; 下料自動允許信號
L3672  ; 下料測試允許信號
L3674  ; 回流測試允許信號
L3812  ; 電熱13  冷卻完成
L3813  ; 電熱14  冷卻完成
L3814  ; 電熱15  冷卻完成
L3815  ; 電熱16  冷卻完成
L3832  ; IRA13   冷卻完成
L3833  ; IRA14   冷卻完成
L3834  ; IRA15   冷卻完成
L3835  ; IRA16   冷卻完成
L3852  ; IRB13   冷卻完成
L3853  ; IRB14   冷卻完成
L3854  ; IRB15   冷卻完成
L3855  ; IRB16   冷卻完成
L3940  ; 溫度到達IRB01
L4002  ; 出料爐體段  警報異常
L4003  ; 出料段  警報異常
L4004  ; 烘烤段  警報異常
L4011  ; 進料爐體段  警報PLS
L4012  ; 出料爐體段  警報PLS
L4013  ; 出料段  警報PLS
L4030  ; 變頻器  復歸信號
L4040  ; 進料機構允許運轉
L4041  ; 爐體機構允許運轉
L4042  ; 下料機構允許運轉
L4043  ; 出料機構允許運轉
L4044  ; 回流機構允許運轉
L4104  ; 掉框板異常PLS
L4118  ; 伺服马达不在位置上異常PLS
L4302  ; 進料牙叉機構回原點
L4307  ; 進料回流機構回原點
L4312  ; 出料牙叉機構回原點
L4313  ; 出料手臂機構回原點
L4317  ; 出料回流機構回原點
L4401  ; 伺服機構在位置上
L4638  ; 進料分流左側旋轉定點光電
L4790  ; 出料手臂機構有板原點
L4791  ; 出料手臂機構無板原點
L7777  ; test
T7  ; 手動進料輸送停止延遲
T14  ; 手動進料手臂下夾板  夾延遲
T15  ; 手動進料手臂下夾板  放延遲
T107  ; 出料輸送變頻器停止延遲
T193  ; 冷卻溫度到達2延遲
T212  ; 第13槽  循環風車SW延遲
T213  ; 第14槽  循環風車SW延遲
T214  ; 第15槽  循環風車SW延遲
T215  ; 第16槽  循環風車SW延遲
T216  ; 第17槽  循環風車SW延遲
T217  ; 第18槽  循環風車SW延遲
T218  ; 第19槽  循環風車SW延遲
T219  ; 第20槽  循環風車SW延遲
T252  ; 第13槽  電熱SW  延遲
T253  ; 第14槽  電熱SW  延遲
T254  ; 第15槽  電熱SW  延遲
T255  ; 第16槽  電熱SW  延遲
T256  ; 第17槽  電熱SW  延遲
T257  ; 第18槽  電熱SW  延遲
T258  ; 第19槽  電熱SW  延遲
T259  ; 第20槽  電熱SW  延遲
T272  ; 第13槽  IRA SW  延遲
T273  ; 第14槽  IRA SW  延遲
T274  ; 第15槽  IRA SW  延遲
T275  ; 第16槽  IRA SW  延遲
T276  ; 第17槽  IRA SW  延遲
T277  ; 第18槽  IRA SW  延遲
T278  ; 第19槽  IRA SW  延遲
T279  ; 第20槽  IRA SW  延遲
T292  ; 第13槽  IRB SW  延遲
T293  ; 第14槽  IRB SW  延遲
T294  ; 第15槽  IRB SW  延遲
T295  ; 第16槽  IRB SW  延遲
T296  ; 第17槽  IRB SW  延遲
T297  ; 第18槽  IRB SW  延遲
T298  ; 第19槽  IRB SW  延遲
T299  ; 第20槽  IRB SW  延遲
T314  ; 自動進料手臂下夾板  夾延遲
T315  ; 自動進料手臂下夾板  放延遲
T318  ; 自動進料回流檔框1上昇延遲
T520  ; 進料擋板原點延遲
T521  ; 進料平台原點延遲
T522  ; 進料手臂內外原點
T523  ; 進料手臂夾爪原點
T525  ; 進料伺服機構要求回原點
T529  ; 進料回流機構要求回原點延遲
T638  ; 進料分流左側旋轉定點光電延遲
T817  ; 出料回流機構要求回原點延遲
T830  ; 出料牙插原點延遲
T831  ; 出料牙插夾爪原點延遲
T832  ; 出料手臂內外原點延遲
T833  ; 出料手臂夾爪原點延遲
T835  ; 出料伺服機構要求回原點延遲
T1003  ; Unload_ CC-Link Delay
T1026  ; 出料手臂至校正位置手動TM
T1055  ; SECS_USE開機延遲一秒
T1083  ; 下料伺服機構無歸零要求
T1093  ; 下料伺服機構無回原點訊號
T1103  ; 進料整板啟動延遲
T1123  ; 進料整板位置04延遲
T1124  ; 進料整板位置05延遲
T1125  ; 進料整板位置06延遲
T1126  ; 進料整板位置07延遲
T1127  ; 進料整板位置08延遲
T1128  ; 進料整板位置09延遲
T1129  ; 進料整板位置10延遲
T1153  ; 進料整板位置自動往  位置04
T1154  ; 進料整板位置自動往  位置05
T1155  ; 進料整板位置自動往  位置06
T1156  ; 進料整板位置自動往  位置07
T1157  ; 進料整板位置自動往  位置08
T1158  ; 進料整板位置自動往  位置09
T1159  ; 進料整板位置自動往  位置10
T1170  ; 進料整板自動往  位置01
T1171  ; 進料整板自動往  位置02
T1172  ; 進料整板自動往  位置03
T1173  ; 進料整板自動往  位置04
T1174  ; 進料整板自動往  位置05
T1175  ; 進料整板自動往  位置06
T1176  ; 進料整板自動往  位置07
T1177  ; 進料整板自動往  位置08
T1178  ; 進料整板自動往  位置09
T1179  ; 進料整板自動往  位置10
T1180  ; 允許進料整板拍板位置01延遲*
T1181  ; 允許進料整板拍板位置02延遲*
T1190  ; 允許進料整板歸位延遲*
T1191  ; 允許進料整板拍板延遲*
T1203  ; 牙插移載啟動延遲
T1222  ; 牙插移載位置03延遲
T1223  ; 牙插移載位置04延遲
T1224  ; 牙插移載位置05延遲
T1225  ; 牙插移載位置06延遲
T1226  ; 牙插移載位置07延遲
T1227  ; 牙插移載位置08延遲
T1228  ; 牙插移載位置09延遲
T1229  ; 牙插移載位置10延遲
T1252  ; 牙插移載位置自動往  位置03
T1253  ; 牙插移載位置自動往  位置04
T1254  ; 牙插移載位置自動往  位置05
T1255  ; 牙插移載位置自動往  位置06
T1256  ; 牙插移載位置自動往  位置07
T1257  ; 牙插移載位置自動往  位置08
T1258  ; 牙插移載位置自動往  位置09
T1259  ; 牙插移載位置自動往  位置10
T1270  ; 牙插移載自動往  位置01
T1271  ; 牙插移載自動往  位置02
T1272  ; 牙插移載自動往  位置03
T1273  ; 牙插移載自動往  位置04
T1274  ; 牙插移載自動往  位置05
T1275  ; 牙插移載自動往  位置06
T1276  ; 牙插移載自動往  位置07
T1277  ; 牙插移載自動往  位置08
T1278  ; 牙插移載自動往  位置09
T1279  ; 牙插移載自動往  位置10
T1290  ; 牙插移載自動往  位置01*
T1403  ; 進手臂取手啟動延遲
T1422  ; 進手臂取手位置03延遲
T1423  ; 進手臂取手位置04延遲
T1424  ; 進手臂取手位置05延遲
T1425  ; 進手臂取手位置06延遲
T1426  ; 進手臂取手位置07延遲
T1427  ; 進手臂取手位置08延遲
T1428  ; 進手臂取手位置09延遲
T1429  ; 進手臂取手位置10延遲
T1452  ; 進手臂取手位置自動往  位置03
T1453  ; 進手臂取手位置自動往  位置04
T1454  ; 進手臂取手位置自動往  位置05
T1455  ; 進手臂取手位置自動往  位置06
T1456  ; 進手臂取手位置自動往  位置07
T1457  ; 進手臂取手位置自動往  位置08
T1458  ; 進手臂取手位置自動往  位置09
T1459  ; 進手臂取手位置自動往  位置10
T1470  ; 進手臂取手自動往  位置01
T1471  ; 進手臂取手自動往  位置02
T1472  ; 進手臂取手自動往  位置03
T1473  ; 進手臂取手自動往  位置04
T1474  ; 進手臂取手自動往  位置05
T1475  ; 進手臂取手自動往  位置06
T1476  ; 進手臂取手自動往  位置07
T1477  ; 進手臂取手自動往  位置08
T1478  ; 進手臂取手自動往  位置09
T1479  ; 進手臂取手自動往  位置10
T1481  ; 允許托框昇降下降位置01延遲*
T1503  ; 進料托框昇降啟動延遲
T1524  ; 進料托框昇降位置05延遲
T1525  ; 進料托框昇降位置06延遲
T1526  ; 進料托框昇降位置07延遲
T1527  ; 進料托框昇降位置08延遲
T1528  ; 進料托框昇降位置09延遲
T1529  ; 進料托框昇降位置10延遲
T1554  ; 進料托框昇降位置自動往  位置05
T1555  ; 進料托框昇降位置自動往  位置06
T1556  ; 進料托框昇降位置自動往  位置07
T1557  ; 進料托框昇降位置自動往  位置08
T1558  ; 進料托框昇降位置自動往  位置09
T1559  ; 進料托框昇降位置自動往  位置10
T1570  ; 進料托框昇降自動往  位置01
T1571  ; 進料托框昇降自動往  位置02
T1572  ; 進料托框昇降自動往  位置03
T1573  ; 進料托框昇降自動往  位置04
T1574  ; 進料托框昇降自動往  位置05
T1575  ; 進料托框昇降自動往  位置06
T1576  ; 進料托框昇降自動往  位置07
T1577  ; 進料托框昇降自動往  位置08
T1578  ; 進料托框昇降自動往  位置09
T1579  ; 進料托框昇降自動往  位置10
T1580  ; 允許回流移載往出料延遲*
T1581  ; 回流移載任一上昇延遲*
T1582  ; 回流移載昇降定位延遲*
T1583  ; 回流移載昇降無動作延遲*
T1590  ; 回流托架上昇允許移載位置02延遲*
T1591  ; 回流托架1上昇允許移載位置02延遲*
T1592  ; 回流托架2上昇允許移載位置02延遲*
T1593  ; 回流托架3上昇允許移載位置02延遲*
T1594  ; 回流托架4上昇允許移載位置02延遲*
T1595  ; 回流托架5上昇允許移載位置02延遲*
T1596  ; 回流托架6上昇允許移載位置02延遲*
T1597  ; 回流托架7上昇允許移載位置02延遲*
T1603  ; 進左開爪啟動延遲
T1625  ; 進左開爪位置06延遲
T1626  ; 進左開爪位置07延遲
T1627  ; 進左開爪位置08延遲
T1628  ; 進左開爪位置09延遲
T1629  ; 進左開爪位置10延遲
T1655  ; 進左開爪位置自動往  位置06
T1656  ; 進左開爪位置自動往  位置07
T1657  ; 進左開爪位置自動往  位置08
T1658  ; 進左開爪位置自動往  位置09
T1659  ; 進左開爪位置自動往  位置10
T1670  ; 進左開爪自動往  位置01
T1671  ; 進左開爪自動往  位置02
T1672  ; 進左開爪自動往  位置03
T1673  ; 進左開爪自動往  位置04
T1674  ; 進左開爪自動往  位置05
T1675  ; 進左開爪自動往  位置06
T1676  ; 進左開爪自動往  位置07
T1677  ; 進左開爪自動往  位置08
T1678  ; 進左開爪自動往  位置09
T1679  ; 進左開爪自動往  位置10
T1703  ; 進右開爪啟動延遲
T1725  ; 進右開爪位置06延遲
T1726  ; 進右開爪位置07延遲
T1727  ; 進右開爪位置08延遲
T1728  ; 進右開爪位置09延遲
T1729  ; 進右開爪位置10延遲
T1755  ; 進右開爪位置自動往  位置06
T1756  ; 進右開爪位置自動往  位置07
T1757  ; 進右開爪位置自動往  位置08
T1758  ; 進右開爪位置自動往  位置09
T1759  ; 進右開爪位置自動往  位置10
T1770  ; 進右開爪自動往  位置01
T1771  ; 進右開爪自動往  位置02
T1772  ; 進右開爪自動往  位置03
T1773  ; 進右開爪自動往  位置04
T1774  ; 進右開爪自動往  位置05
T1775  ; 進右開爪自動往  位置06
T1776  ; 進右開爪自動往  位置07
T1777  ; 進右開爪自動往  位置08
T1778  ; 進右開爪自動往  位置09
T1779  ; 進右開爪自動往  位置10
T2036  ; CCD 對位延遲
T2047  ; Y-20-OK
T2048  ; X-20-OK
T2056  ; CCD 對位延遲2再觸發1
T2057  ; CCD 對位延遲2再觸發2
T2103  ; 分流前取框啟動延遲
T2123  ; 分流前取框位置04延遲
T2124  ; 分流前取框位置05延遲
T2125  ; 分流前取框位置06延遲
T2126  ; 分流前取框位置07延遲
T2127  ; 分流前取框位置08延遲
T2128  ; 分流前取框位置09延遲
T2129  ; 分流前取框位置10延遲
T2153  ; 分流前取框位置自動往  位置04
T2154  ; 分流前取框位置自動往  位置05
T2155  ; 分流前取框位置自動往  位置06
T2156  ; 分流前取框位置自動往  位置07
T2157  ; 分流前取框位置自動往  位置08
T2158  ; 分流前取框位置自動往  位置09
T2159  ; 分流前取框位置自動往  位置10
T2170  ; 分流前取框自動往  位置01
T2171  ; 分流前取框自動往  位置02
T2172  ; 分流前取框自動往  位置03
T2173  ; 分流前取框自動往  位置04
T2174  ; 分流前取框自動往  位置05
T2175  ; 分流前取框自動往  位置06
T2176  ; 分流前取框自動往  位置07
T2177  ; 分流前取框自動往  位置08
T2178  ; 分流前取框自動往  位置09
T2179  ; 分流前取框自動往  位置10
T2203  ; 合流後掛框啟動延遲
T2223  ; 合流後掛框位置04延遲
T2224  ; 合流後掛框位置05延遲
T2225  ; 合流後掛框位置06延遲
T2226  ; 合流後掛框位置07延遲
T2227  ; 合流後掛框位置08延遲
T2228  ; 合流後掛框位置09延遲
T2229  ; 合流後掛框位置10延遲
T2253  ; 合流後掛框位置自動往  位置04
T2254  ; 合流後掛框位置自動往  位置05
T2255  ; 合流後掛框位置自動往  位置06
T2256  ; 合流後掛框位置自動往  位置07
T2257  ; 合流後掛框位置自動往  位置08
T2258  ; 合流後掛框位置自動往  位置09
T2259  ; 合流後掛框位置自動往  位置10
T2270  ; 合流後掛框自動往  位置01
T2271  ; 合流後掛框自動往  位置02
T2272  ; 合流後掛框自動往  位置03
T2273  ; 合流後掛框自動往  位置04
T2274  ; 合流後掛框自動往  位置05
T2275  ; 合流後掛框自動往  位置06
T2276  ; 合流後掛框自動往  位置07
T2277  ; 合流後掛框自動往  位置08
T2278  ; 合流後掛框自動往  位置09
T2279  ; 合流後掛框自動往  位置10
T2625  ; 允許配方寫入延遲-TM
T3103  ; 出手臂取手啟動延遲
T3123  ; 出手臂取手位置04延遲
T3124  ; 出手臂取手位置05延遲
T3125  ; 出手臂取手位置06延遲
T3126  ; 出手臂取手位置07延遲
T3127  ; 出手臂取手位置08延遲
T3128  ; 出手臂取手位置09延遲
T3129  ; 出手臂取手位置10延遲
T3153  ; 出手臂取手位置自動往  位置04
T3154  ; 出手臂取手位置自動往  位置05
T3155  ; 出手臂取手位置自動往  位置06
T3156  ; 出手臂取手位置自動往  位置07
T3157  ; 出手臂取手位置自動往  位置08
T3158  ; 出手臂取手位置自動往  位置09
T3159  ; 出手臂取手位置自動往  位置10
T3170  ; 出手臂取手自動往  位置01
T3171  ; 出手臂取手自動往  位置02
T3172  ; 出手臂取手自動往  位置03
T3173  ; 出手臂取手自動往  位置04
T3174  ; 出手臂取手自動往  位置05
T3175  ; 出手臂取手自動往  位置06
T3176  ; 出手臂取手自動往  位置07
T3177  ; 出手臂取手自動往  位置08
T3178  ; 出手臂取手自動往  位置09
T3179  ; 出手臂取手自動往  位置10
T3203  ; 出料托框昇降啟動延遲
T3225  ; 出料托框昇降位置06延遲
T3226  ; 出料托框昇降位置07延遲
T3227  ; 出料托框昇降位置08延遲
T3228  ; 出料托框昇降位置09延遲
T3229  ; 出料托框昇降位置10延遲
T3255  ; 出料托框昇降位置自動往  位置06
T3256  ; 出料托框昇降位置自動往  位置07
T3257  ; 出料托框昇降位置自動往  位置08
T3258  ; 出料托框昇降位置自動往  位置09
T3270  ; 出料托框昇降自動往  位置01
T3271  ; 出料托框昇降自動往  位置02
T3272  ; 出料托框昇降自動往  位置03
T3273  ; 出料托框昇降自動往  位置04
T3274  ; 出料托框昇降自動往  位置05
T3275  ; 出料托框昇降自動往  位置06
T3276  ; 出料托框昇降自動往  位置07
T3277  ; 出料托框昇降自動往  位置08
T3278  ; 出料托框昇降自動往  位置09
T3279  ; 出料托框昇降自動往  位置10
T3303  ; 出左開夾啟動延遲
T3325  ; 出左開夾位置06延遲
T3326  ; 出左開夾位置07延遲
T3327  ; 出左開夾位置08延遲
T3328  ; 出左開夾位置09延遲
T3329  ; 出左開夾位置10延遲
T3355  ; 出左開夾位置自動往  位置06
T3356  ; 出左開夾位置自動往  位置07
T3357  ; 出左開夾位置自動往  位置08
T3358  ; 出左開夾位置自動往  位置09
T3359  ; 出左開夾位置自動往  位置10
T3370  ; 出左開夾自動往  位置01
T3371  ; 出左開夾自動往  位置02
T3372  ; 出左開夾自動往  位置03
T3373  ; 出左開夾自動往  位置04
T3374  ; 出左開夾自動往  位置05
T3375  ; 出左開夾自動往  位置06
T3376  ; 出左開夾自動往  位置07
T3377  ; 出左開夾自動往  位置08
T3378  ; 出左開夾自動往  位置09
T3379  ; 出左開夾自動往  位置10
T3403  ; 出右開夾啟動延遲
T3425  ; 出右開夾位置06延遲
T3426  ; 出右開夾位置07延遲
T3427  ; 出右開夾位置08延遲
T3428  ; 出右開夾位置09延遲
T3429  ; 出右開夾位置10延遲
T3455  ; 出右開夾位置自動往  位置06
T3456  ; 出右開夾位置自動往  位置07
T3457  ; 出右開夾位置自動往  位置08
T3458  ; 出右開夾位置自動往  位置09
T3459  ; 出右開夾位置自動往  位置10
T3470  ; 出右開夾自動往  位置01
T3471  ; 出右開夾自動往  位置02
T3472  ; 出右開夾自動往  位置03
T3473  ; 出右開夾自動往  位置04
T3474  ; 出右開夾自動往  位置05
T3475  ; 出右開夾自動往  位置06
T3476  ; 出右開夾自動往  位置07
T3477  ; 出右開夾自動往  位置08
T3478  ; 出右開夾自動往  位置09
T3479  ; 出右開夾自動往  位置10
T3503  ; 出板牙插移載啟動延遲
T3523  ; 出板牙插移載位置04延遲
T3524  ; 出板牙插移載位置05延遲
T3525  ; 出板牙插移載位置06延遲
T3526  ; 出板牙插移載位置07延遲
T3527  ; 出板牙插移載位置08延遲
T3528  ; 出板牙插移載位置09延遲
T3529  ; 出板牙插移載位置10延遲
T3553  ; 出板牙插移載位置自動往  位置04
T3554  ; 出板牙插移載位置自動往  位置05
T3555  ; 出板牙插移載位置自動往  位置06
T3556  ; 出板牙插移載位置自動往  位置07
T3557  ; 出板牙插移載位置自動往  位置08
T3558  ; 出板牙插移載位置自動往  位置09
T3559  ; 出板牙插移載位置自動往  位置10
T3570  ; 出板牙插移載自動往  位置01
T3571  ; 出板牙插移載自動往  位置02
T3572  ; 出板牙插移載自動往  位置03
T3573  ; 出板牙插移載自動往  位置04
T3574  ; 出板牙插移載自動往  位置05
T3575  ; 出板牙插移載自動往  位置06
T3576  ; 出板牙插移載自動往  位置07
T3577  ; 出板牙插移載自動往  位置08
T3578  ; 出板牙插移載自動往  位置09
T3579  ; 出板牙插移載自動往  位置10
T3900  ; 出料牙叉上層    上定點異常延遲
T3901  ; 出料牙叉上層    下定點異常延遲
T3902  ; 出料牙叉下層    上定點異常延遲
T3903  ; 出料牙叉下層    下定點異常延遲
T4002  ; 進料牙叉機構回原點延遲
T4007  ; 進料回流機構回原點延遲
T4012  ; 出料牙叉機構回原點延遲
T4013  ; 出料手臂機構回原點延遲
T4017  ; 出料回流機構回原點延遲
T4052  ; 進料牙叉機構回原點逾時
T4057  ; 進料回流機構回原點逾時
T4062  ; 出料牙叉機構回原點逾時
T4063  ; 出料手臂機構回原點逾時
T4067  ; 出料回流機構回原點逾時
T4148  ; 進料輸送入口光電異常延遲
T4149  ; 進料輸送減速光電異常延遲
T4209  ; 合流右_旋轉定點異常延遲
T4300  ; 第1槽 OTP超溫延遲
T4301  ; 第2槽 OTP超溫延遲
T4302  ; 第3槽 OTP超溫延遲
T4303  ; 第4槽 OTP超溫延遲
T4304  ; 第5槽 OTP超溫延遲
T4305  ; 第6槽 OTP超溫延遲
T4306  ; 第7槽 OTP超溫延遲
T4307  ; 第8槽 OTP超溫延遲
T4308  ; 第9槽 OTP超溫延遲
T4309  ; 第10槽 OTP超溫延遲
T4310  ; 第11槽 OTP超溫延遲
T4311  ; 第12槽 OTP超溫延遲
T4312  ; 第13槽 OTP超溫延遲
T4313  ; 第14槽 OTP超溫延遲
T4314  ; 第15槽 OTP超溫延遲
T4315  ; 第16槽 OTP超溫延遲
T4320  ; 第1槽  IRA OTP 超溫延遲
T4321  ; 第2槽  IRA OTP 超溫延遲
T4322  ; 第3槽  IRA OTP 超溫延遲
T4323  ; 第4槽  IRA OTP 超溫延遲
T4324  ; 第5槽  IRA OTP 超溫延遲
T4325  ; 第6槽  IRA OTP 超溫延遲
T4326  ; 第7槽  IRA OTP 超溫延遲
T4327  ; 第8槽  IRA OTP 超溫延遲
T4328  ; 第9槽  IRA OTP 超溫延遲
T4329  ; 第10槽  IRA OTP 超溫延遲
T4330  ; 第11槽  IRA OTP 超溫延遲
T4331  ; 第12槽  IRA OTP 超溫延遲
T4332  ; 第13槽  IRA OTP 超溫延遲
T4333  ; 第14槽  IRA OTP 超溫延遲
T4334  ; 第15槽  IRA OTP 超溫延遲
T4335  ; 第16槽  IRA OTP 超溫延遲
T4340  ; 第1槽  IRB OTP 超溫延遲
T4341  ; 第2槽  IRB OTP 超溫延遲
T4342  ; 第3槽  IRB OTP 超溫延遲
T4343  ; 第4槽  IRB OTP 超溫延遲
T4344  ; 第5槽  IRB OTP 超溫延遲
T4345  ; 第6槽  IRB OTP 超溫延遲
T4346  ; 第7槽  IRB OTP 超溫延遲
T4347  ; 第8槽  IRB OTP 超溫延遲
T4348  ; 第9槽  IRB OTP 超溫延遲
T4349  ; 第10槽  IRB OTP 超溫延遲
T4350  ; 第11槽  IRB OTP 超溫延遲
T4351  ; 第12槽  IRB OTP 超溫延遲
T4352  ; 第13槽  IRB OTP 超溫延遲
T4353  ; 第14槽  IRB OTP 超溫延遲
T4354  ; 第15槽  IRB OTP 超溫延遲
T4355  ; 第16槽  IRB OTP 超溫延遲
T4360  ; 第1槽風車馬達異常延遲
T4361  ; 第2槽風車馬達異常延遲
T4362  ; 第3槽風車馬達異常延遲
T4363  ; 第4槽風車馬達異常延遲
T4364  ; 第5槽風車馬達異常延遲
T4365  ; 第6槽風車馬達異常延遲
T4366  ; 第7槽風車馬達異常延遲
T4367  ; 第8槽風車馬達異常延遲
T4372  ; 第13槽風車馬達異常延遲
T4373  ; 第14槽風車馬達異常延遲
T4374  ; 第15槽風車馬達異常延遲
T4375  ; 第16槽風車馬達異常延遲
T4380  ; 第1槽風車馬達過載延遲
T4381  ; 第2槽風車馬達過載延遲
T4382  ; 第3槽風車馬達過載延遲
T4383  ; 第4槽風車馬達過載延遲
T4384  ; 第5槽風車馬達過載延遲
T4385  ; 第6槽風車馬達過載延遲
T4386  ; 第7槽風車馬達過載延遲
T4387  ; 第8槽風車馬達過載延遲
T4388  ; 第9槽風車馬達過載延遲
T4389  ; 第10槽風車馬達過載延遲
T4390  ; 第11槽風車馬達過載延遲
T4391  ; 第12槽風車馬達過載延遲
T4392  ; 第13槽風車馬達過載延遲
T4393  ; 第14槽風車馬達過載延遲
T4394  ; 第15槽風車馬達過載延遲
T4395  ; 第16槽風車馬達過載延遲
T4420  ; 第01段  低溫延遲
T4421  ; 第02段  低溫延遲
T4422  ; 第03段  低溫延遲
T4423  ; 第04段  低溫延遲
T4424  ; 第05段  低溫延遲
T4425  ; 第06段  低溫延遲
T4426  ; 第07段  低溫延遲
T4427  ; 第08段  低溫延遲
T4428  ; 第09段  低溫延遲
T4429  ; 第10段  低溫延遲
T4680  ; 進料整板歸零要求異常延遲
T4681  ; 取板牙插歸零要求異常延遲
T4683  ; 進料手臂取手歸零要求異常延遲
T4684  ; 進料托框昇降歸零要求異常延遲
T4685  ; 進左開夾歸零要求異常延遲
T4686  ; 進右開夾歸零要求異常延遲
T4687  ; 分流前取框歸零要求異常延遲
T4688  ; 出板牙插歸零要求異常延遲
T4690  ; 出料手臂取手歸零要求異常延遲
T4691  ; 出料托框昇降歸零要求異常延遲
T4692  ; 出左開夾歸零要求異常延遲
T4693  ; 出右開夾歸零要求異常延遲
T4694  ; 合流後掛框歸零要求異常延遲
D6  ; 進料人機畫頁狀態區
D8  ; 進料人機畫頁變更顯示
D12  ; 進料HMI 時間修改日
D13  ; 進料HMI 時間修改時分
D22  ; 出料人機日期年BCD
D23  ; 出料人機日期月BCD
D24  ; 出料人機日期日BCD
D25  ; 出料人機日期時分BCD
D26  ; 出料人機畫頁狀態區
D28  ; 出料人機畫頁變更顯示
D30  ; 出料HMI 時間修改年
D31  ; 出料HMI 時間修改月
D32  ; 出料HMI 時間修改日
D33  ; 出料HMI 時間修改時分
D36  ; 出料視窗控制
D37  ; 出料視窗登錄號碼
D38  ; 出料視窗顯示X 座標
D39  ; 出料視窗顯示Y 座標
D60  ; Q62DAN  模組異常碼
D93  ; 單邊槽數設定4
D97  ; 進料人機權限密碼
D98  ; 出料人機權限密碼
D901  ; 進料手臂取板補償X軸
D903  ; 進料手臂取板補償Y軸
D905  ; 進料手臂取板補償Z軸
D906  ; 進料手臂取板補償θ軸
D907  ; 進料手臂取板補償θ軸
D1039  ; #09啟動位置選擇
D1065  ; 位置有板顯示
D1081  ; 進料框架來源尺寸長0.000
D1083  ; 進料分流左側框架尺寸    長0.000
D1085  ; 進料分流右側框架尺寸    長0.000
D1101  ; 整板現在位置
D1103  ; 整板現在速度
D1116  ; 小板移載位置01
D1201  ; 牙插移載現在位置
D1203  ; 牙插移載現在速度
D1401  ; 進手臂取手現在位置
D1403  ; 進手臂取手現在速度
D1416  ; 大板模式拉撐位置
D1417  ; 大板模式拉撐位置
D1418  ; 小板模式拉撐位置
D1419  ; 小板模式拉撐位置
D1501  ; 進料托框昇降現在位置
D1503  ; 進料托框昇降現在速度
D1601  ; 進左開爪現在位置
D1603  ; 進左開爪現在速度
D1701  ; 進右開爪現在位置
D1703  ; 進右開爪現在速度
D1901  ; X_Float
D1903  ; No.1 X_ Float
D1905  ; No.1 Y_ Float
D1907  ; No.2 X_ Float
D1909  ; No.2 Y_ Float
D1911  ; Y2 - Y1 Float
D1913  ; X2 - X1 Float
D1915  ; X - X1  Float
D1917  ; Y2 - Y1 --------X2 - X1
D1919  ; ========================
D1930  ; X_Float  類比輸入
D1931  ; X_Float  類比輸入
D1933  ; No.1 X_ Float
D1935  ; No.1 Y_ Float
D1937  ; No.2 X_ Float
D1939  ; No.2 Y_ Float
D2071  ; 加熱中  視窗
D2073  ; 冷卻中  視窗
D2080  ; 步進倒數時間SEC
D2081  ; 烘烤時間秒鐘
D2082  ; 烘烤時間秒鐘
D2083  ; 步進間隔時間SEC 整數
D2084  ; 步進間隔時間SEC 整數
D2085  ; 步進間隔時間SEC 餘數
D2086  ; 步進間隔時間SEC 餘數
D2088  ; 步進倒數時間SEC
D2090  ; 步進倒數時間顯示整數
D2091  ; 步進倒數時間顯示餘數
D2092  ; 步進倒數時間顯示餘數
D2101  ; 分流前取框現在位置
D2103  ; 分流前取框現在速度
D2201  ; 合流後掛框現在位置
D2203  ; 合流後掛框現在速度
D2501  ; RB1人機手臂印刷取板點(補償)X_SV
D2502  ; RB1人機手臂取板點(補償)Y_SV
D2503  ; RB1人機手臂取板點(補償)Z_SV
D2504  ; RB1人機接駁放板點(前後補償)X_SV
D2505  ; RB1人機接駁放板點(左右補償)Y_SV
D2506  ; RB1人機接駁放板點(升降補償)Z_SV
D2507  ; RB1人機檢查取板點(前後補償)X_SV
D2508  ; RB人機檢查取板點(左右補償)Y_SV
D2509  ; RB1人機檢查取板點(升降補償)Z_SV
D2510  ; R0B0T1實際板長-最大板長(Y)商數
D2511  ; R0B0T1實際板長-最大板長(Y)餘數
D2514  ; R0B0T1實際板寬-最小板寬(Y)商數
D2515  ; R0B0T1實際板寬-最小板寬(Y)餘數
D2518  ; R0B0T1機器人教點尺寸-最大板寬
D2522  ; R0B0T1人機手臂取板點(補償)Y
D2526  ; R0B0T1人機手臂放板點(補償)Z
D2531  ; RB1人機檢查放板點(前後補償)X_SV
D2532  ; RB人機檢查放板點(左右補償)Y_SV
D2533  ; RB1人機檢查放板點(升降補償)Z_SV
D2653  ; CCD 重置ˋ次數
D2700  ; CCD>>PLC心跳每秒切替
D2704  ; CCD>>PLCY補償   小數3位 *1000
D2706  ; CCD>>PLCT補償   小數3位 *1000
D2728  ; CCD>>PLC板寬
D2730  ; CCD>>PLC板長
D2731  ; CCD_X軸+補正(0.00 mm)
D2732  ; CCD_X軸-補正(0.00 mm)
D2733  ; CCD_Y軸+補正(0.00 mm)
D2734  ; CCD_Y軸-補正(0.00 mm)
D2735  ; CCD_T軸+補正(0.00 mm)
D2736  ; CCD_T軸-補正(0.00 mm)
D2801  ; CCD_X補償+偏差補償_整數
D2802  ; CCD_X補償+偏差補償_小數
D2803  ; CCD_X補償+偏差補償_小數
D2811  ; CCD_Y補償+偏差補償_整數
D2812  ; CCD_Y補償+偏差補償_小數
D2813  ; CCD_Y補償+偏差補償_小數
D2821  ; CCD_T補償+偏差補償_整數
D2822  ; CCD_T補償+偏差補償_小數
D2823  ; CCD_T補償+偏差補償_小數
D2831  ; 人機Z補償_整數
D2832  ; 人機Z補償_小數
D2833  ; 人機Z補償_小數
D2900  ; 人機出料取板偏差補償整數X
D2901  ; 人機出料取板偏差補償整數X
D2903  ; 人機出料取板偏差補償整數X給RB
D2904  ; 人機出料取板偏差補償小數XX給RB
D2905  ; 人機出料取板偏差補償小數XX給RB
D2910  ; 人機出料取板偏差補償整數Y
D2911  ; 人機出料取板偏差補償整數Y
D2913  ; 人機出料取板偏差補償整數Y給RB
D2914  ; 人機出料取板偏差補償小數YY給RB
D2915  ; 人機出料取板偏差補償小數YY給RB
D2920  ; 人機出料取板偏差補償整數Z
D2921  ; 人機出料取板偏差補償整數Z
D2923  ; 人機出料取板偏差補償整數Z給RB
D2924  ; 人機出料取板偏差補償小數ZZ給RB
D2925  ; 人機出料取板偏差補償小數ZZ給RB
D2951  ; 人機出料放板偏差補償整數X
D2953  ; 人機出料放板偏差補償整數X給RB
D2955  ; 人機出料放板偏差補償小數XX給RB
D2961  ; 人機出料放板偏差補償整數Y
D2963  ; 人機出料放板偏差補償整數Y給RB
D2965  ; 人機出料放板偏差補償小數YY給RB
D2971  ; 人機出料放板偏差補償整數Z
D2973  ; 人機出料放板偏差補償整數Z給RB
D2975  ; 人機出料放板偏差補償小數ZZ給RB
D2981  ; 人機出料放板偏差補償整數T
D2983  ; 人機出料放板偏差補償整數T給RB
D2984  ; 人機出料放板偏差補償小數TT給RB
D2985  ; 人機出料放板偏差補償小數TT給RB
D3101  ; 出手臂取手現在位置
D3103  ; 出手臂取手現在速度
D3201  ; 出料托框昇降現在位置
D3203  ; 出料托框昇降現在速度
D3301  ; 出左開夾現在位置
D3303  ; 出左開夾現在速度
D3401  ; 出右開夾現在位置
D3403  ; 出右開夾現在速度
D3501  ; 出板牙插移載現在位置
D3503  ; 出板牙插移載現在速度
D4003  ; 左側爐內位置03  尺寸
D4004  ; 左側爐內位置04  尺寸
D4005  ; 左側爐內位置05  尺寸
D4006  ; 左側爐內位置06  尺寸
D4007  ; 左側爐內位置07  尺寸
D4008  ; 左側爐內位置08  尺寸
D4009  ; 左側爐內位置09  尺寸
D4010  ; 左側爐內位置10  尺寸
D4011  ; 左側爐內位置11  尺寸
D4012  ; 左側爐內位置12  尺寸
D4013  ; 左側爐內位置13  尺寸
D4014  ; 左側爐內位置14  尺寸
D4015  ; 左側爐內位置15  尺寸
D4016  ; 左側爐內位置16  尺寸
D4017  ; 左側爐內位置17  尺寸
D4018  ; 左側爐內位置18  尺寸
D4019  ; 左側爐內位置19  尺寸
D4020  ; 左側爐內位置20  尺寸
D4051  ; 左側爐內位置01  有板
D4052  ; 左側爐內位置02  有板
D4053  ; 左側爐內位置03  有板
D4054  ; 左側爐內位置04  有板
D4055  ; 左側爐內位置05  有板
D4056  ; 左側爐內位置06  有板
D4057  ; 左側爐內位置07  有板
D4058  ; 左側爐內位置08  有板
D4059  ; 左側爐內位置09  有板
D4060  ; 左側爐內位置10  有板
D4061  ; 左側爐內位置11  有板
D4062  ; 左側爐內位置12  有板
D4063  ; 左側爐內位置13  有板
D4064  ; 左側爐內位置14  有板
D4065  ; 左側爐內位置15  有板
D4066  ; 左側爐內位置16  有板
D4067  ; 左側爐內位置17  有板
D4068  ; 左側爐內位置18  有板
D4069  ; 左側爐內位置19  有板
D4070  ; 左側爐內位置20  有板
D4080  ; 左側爐內板數+1
D4091  ; 出料合流左側框架有板
D4103  ; 右側爐內位置03  尺寸
D4104  ; 右側爐內位置04  尺寸
D4105  ; 右側爐內位置05  尺寸
D4106  ; 右側爐內位置06  尺寸
D4107  ; 右側爐內位置07  尺寸
D4108  ; 右側爐內位置08  尺寸
D4109  ; 右側爐內位置09  尺寸
D4110  ; 右側爐內位置10  尺寸
D4111  ; 右側爐內位置11  尺寸
D4112  ; 右側爐內位置12  尺寸
D4113  ; 右側爐內位置13  尺寸
D4114  ; 右側爐內位置14  尺寸
D4115  ; 右側爐內位置15  尺寸
D4116  ; 右側爐內位置16  尺寸
D4117  ; 右側爐內位置17  尺寸
D4118  ; 右側爐內位置18  尺寸
D4119  ; 右側爐內位置19  尺寸
D4120  ; 右側爐內位置20  尺寸
D4151  ; 右側爐內位置01  有板
D4152  ; 右側爐內位置02  有板
D4153  ; 右側爐內位置03  有板
D4154  ; 右側爐內位置04  有板
D4155  ; 右側爐內位置05  有板
D4156  ; 右側爐內位置06  有板
D4157  ; 右側爐內位置07  有板
D4158  ; 右側爐內位置08  有板
D4159  ; 右側爐內位置09  有板
D4160  ; 右側爐內位置10  有板
D4161  ; 右側爐內位置11  有板
D4162  ; 右側爐內位置12  有板
D4163  ; 右側爐內位置13  有板
D4164  ; 右側爐內位置14  有板
D4165  ; 右側爐內位置15  有板
D4166  ; 右側爐內位置16  有板
D4167  ; 右側爐內位置17  有板
D4168  ; 右側爐內位置18  有板
D4169  ; 右側爐內位置19  有板
D4170  ; 右側爐內位置20  有板
D4180  ; 右側爐內板數+1
D4191  ; 出料合流右側框架有板
D5001  ; 進料手臂板長設定310~610
D5003  ; 進料手臂板寬設定250~510
D5015  ; 進料手臂取手目標位置暫存
D5021  ; 出料手臂板長設定310~610
D5023  ; 出料手臂板寬設定250~510
D5035  ; 出料手臂取手目標位置暫存
D5051  ; 進料輸送板長設定310~610
D5052  ; 進料輸送板寬設定250~510
D5053  ; 進料輸送板寬設定250~510
D5091  ; 最大板長限制設定#610mm
D5093  ; 最小板長限制設定#310mm
D5100  ; PV H01
D5300  ; PV H01
D5312  ; PV H13
D5313  ; PV H14
D5314  ; PV H15
D5315  ; PV H16
D5316  ; PV H17
D5317  ; PV H18
D5318  ; PV H19
D5319  ; PV H20
D5332  ; PV IRA13
D5333  ; PV IRA14
D5334  ; PV IRA15
D5335  ; PV IRA16
D5336  ; PV IRA17
D5337  ; PV IRA18
D5338  ; PV IRA19
D5339  ; PV IRA20
D5352  ; PV IRB13
D5353  ; PV IRB14
D5354  ; PV IRB15
D5355  ; PV IRB16
D5356  ; PV IRB17
D5357  ; PV IRB18
D5358  ; PV IRB19
D5359  ; PV IRB20
D5391  ; S相電流
D5392  ; KWH 總功率
D5393  ; KWH 總功率
D5412  ; SV H13
D5413  ; SV H14
D5414  ; SV H15
D5415  ; SV H16
D5416  ; SV H17
D5417  ; SV H18
D5418  ; SV H19
D5419  ; SV H20
D5432  ; SV IRA13
D5433  ; SV IRA14
D5434  ; SV IRA15
D5435  ; SV IRA16
D5436  ; SV IRA17
D5437  ; SV IRA18
D5438  ; SV IRA19
D5439  ; SV IRA20
D5452  ; SV IRB13
D5453  ; SV IRB14
D5454  ; SV IRB15
D5455  ; SV IRB16
D5456  ; SV IRB17
D5457  ; SV IRB18
D5458  ; SV IRB19
D5459  ; SV IRB20
D5560  ; 溫度昇溫到達01溫度
D5561  ; 溫度昇溫到達02溫度
D5562  ; 溫度昇溫到達03溫度
D5563  ; 溫度昇溫到達04溫度
D5564  ; 溫度昇溫到達05溫度
D5565  ; 溫度昇溫到達06溫度
D5566  ; 溫度昇溫到達07溫度
D5567  ; 溫度昇溫到達08溫度
D5568  ; 溫度昇溫到達09溫度
D5569  ; 溫度昇溫到達10溫度
D5570  ; 溫度昇溫到達11溫度
D5571  ; 溫度昇溫到達12溫度
D5572  ; 溫度昇溫到達13溫度
D5573  ; 溫度昇溫到達14溫度
D5574  ; 溫度昇溫到達15溫度
D5575  ; 溫度昇溫到達16溫度
D5576  ; 溫度昇溫到達17溫度
D5577  ; 溫度昇溫到達18溫度
D5578  ; 溫度昇溫到達19溫度
D5579  ; 溫度昇溫到達20溫度
D5580  ; 溫度降溫到達01溫度
D5581  ; 溫度降溫到達02溫度
D5582  ; 溫度降溫到達03溫度
D5583  ; 溫度降溫到達04溫度
D5584  ; 溫度降溫到達05溫度
D5585  ; 溫度降溫到達06溫度
D5586  ; 溫度降溫到達07溫度
D5587  ; 溫度降溫到達08溫度
D5588  ; 溫度降溫到達09溫度
D5589  ; 溫度降溫到達10溫度
D5590  ; 溫度降溫到達11溫度
D5591  ; 溫度降溫到達12溫度
D5592  ; 溫度降溫到達13溫度
D5593  ; 溫度降溫到達14溫度
D5594  ; 溫度降溫到達15溫度
D5595  ; 溫度降溫到達16溫度
D5596  ; 溫度降溫到達17溫度
D5597  ; 溫度降溫到達18溫度
D5598  ; 溫度降溫到達19溫度
D5599  ; 溫度降溫到達20溫度
D5701  ; 低溫溫度02
D5702  ; 低溫溫度03
D5703  ; 低溫溫度04
D5704  ; 低溫溫度05
D5705  ; 低溫溫度06
D5706  ; 低溫溫度07
D5707  ; 低溫溫度08
D5708  ; 低溫溫度09
D5709  ; 低溫溫度10
D5710  ; 低溫溫度11
D5711  ; 低溫溫度12
D5712  ; 低溫溫度13
D5713  ; 低溫溫度14
D5714  ; 低溫溫度15
D5715  ; 低溫溫度16
D5716  ; 低溫溫度17
D5717  ; 低溫溫度18
D5718  ; 低溫溫度19
D5719  ; 低溫溫度20
D5721  ; 低溫溫度22
D5722  ; 低溫溫度23
D5723  ; 低溫溫度24
D5724  ; 低溫溫度25
D5725  ; 低溫溫度26
D5726  ; 低溫溫度27
D5727  ; 低溫溫度28
D5801  ; 低溫設定溫度02
D5802  ; 低溫設定溫度03
D5803  ; 低溫設定溫度04
D5804  ; 低溫設定溫度05
D5805  ; 低溫設定溫度06
D5806  ; 低溫設定溫度07
D5807  ; 低溫設定溫度08
D5808  ; 低溫設定溫度09
D5809  ; 低溫設定溫度10
D5810  ; 低溫設定溫度11
D5811  ; 低溫設定溫度12
D5812  ; 低溫設定溫度13
D5813  ; 低溫設定溫度14
D5814  ; 低溫設定溫度15
D5815  ; 低溫設定溫度16
D5816  ; 低溫設定溫度17
D5817  ; 低溫設定溫度18
D5818  ; 低溫設定溫度19
D5819  ; 低溫設定溫度20
D5821  ; 低溫設定溫度22
D5822  ; 低溫設定溫度23
D5823  ; 低溫設定溫度24
D5824  ; 低溫設定溫度25
D5825  ; 低溫設定溫度26
D5826  ; 低溫設定溫度27
D5827  ; 低溫設定溫度28
D5900  ; Length_ Out
D5901  ; Length_ Out
D5902  ; Length_ In
D5903  ; Length_ In
D5904  ; Section No
D5905  ; Section No
D5906  ; Length_S
D5907  ; Length_S
D5908  ; Pitch
D5909  ; Pitch
D5966  ; Outlet  Length
D5967  ; Outlet  Length
D5968  ; Inlet   Length
D5969  ; Inlet   Length
D5971  ; Section No.
D5973  ; Section Length
D5975  ; Frame   Pitch
D5976  ; Heating Frame   No.
D5977  ; Heating Frame   No.
D5979  ; Heating Length
D6101  ; COMMANT 02
D6102  ; COMMANT 03
D6103  ; COMMANT 04
D6104  ; COMMANT 05
D6105  ; COMMANT 06
D6106  ; COMMANT 07
D6107  ; COMMANT 08
D6108  ; COMMANT 09
D6109  ; COMMANT 10
D6110  ; COMMANT 11
D6111  ; COMMANT 12
D6112  ; COMMANT 13
D6113  ; COMMANT 14
D6114  ; COMMANT 15
D6115  ; COMMANT 16
D6116  ; COMMANT 17
D6117  ; COMMANT 18
D6118  ; COMMANT 19
D6119  ; COMMANT 20
D6121  ; 配方設定SV H02
D6122  ; 配方設定SV H03
D6123  ; 配方設定SV H04
D6124  ; 配方設定SV H05
D6125  ; 配方設定SV H06
D6126  ; 配方設定SV H07
D6127  ; 配方設定SV H08
D6128  ; 配方設定SV H09
D6129  ; 配方設定SV H10
D6130  ; 配方設定SV H11
D6131  ; 配方設定SV H12
D6140  ; 配方設定SV IRA01
D6141  ; 配方設定SV IRA02
D6142  ; 配方設定SV IRA03
D6143  ; 配方設定SV IRA04
D6144  ; 配方設定SV IRA05
D6145  ; 配方設定SV IRA06
D6146  ; 配方設定SV IRA07
D6147  ; 配方設定SV IRA08
D6148  ; 配方設定SV IRA09
D6149  ; 配方設定SV IRA10
D6150  ; 配方設定SV IRA11
D6151  ; 配方設定SV IRA12
D6160  ; 配方設定SV IRB01
D6161  ; 配方設定SV IRB02
D6162  ; 配方設定SV IRB03
D6163  ; 配方設定SV IRB04
D6164  ; 配方設定SV IRB05
D6165  ; 配方設定SV IRB06
D6166  ; 配方設定SV IRB07
D6167  ; 配方設定SV IRB08
D6168  ; 配方設定SV IRB09
D6169  ; 配方設定SV IRB10
D6170  ; 配方設定SV IRB11
D6171  ; 配方設定SV IRB12
D6209  ; HMI-配方名稱
D7010  ; Barcode 配方組數
D7121  ; 加熱02  冷卻設定溫度
D7122  ; 加熱03  冷卻設定溫度
D7123  ; 加熱04  冷卻設定溫度
D7124  ; 加熱05  冷卻設定溫度
D7125  ; 加熱06  冷卻設定溫度
D7126  ; 加熱07  冷卻設定溫度
D7127  ; 加熱08  冷卻設定溫度
D7128  ; 加熱09  冷卻設定溫度
D7129  ; 加熱10  冷卻設定溫度
D7160  ; 加熱視窗
D7170  ; 冷卻視窗
D7213  ; 本班產能
D7217  ; 爐內板數
D7219  ; 總產能
D7290  ; 炉内片数
D7291  ; 批次剩余数量
D7303  ; 系統時間年月日01
D7304  ; 系統時間年月日02
D7305  ; 系統時間年月日02
D7306  ; 系統時間年月日03
D7307  ; 系統時間年月日03
D7308  ; 系統時間年月日04
D7309  ; 系統時間年月日04
D7310  ; 系統時間年月日05
D7311  ; 系統時間年月日05
D7312  ; 系統時間年月日06
D7313  ; 系統時間年月日06
D7314  ; 系統時間年月日07
D7315  ; 系統時間年月日07
D7316  ; 系統時間年月日08
D7317  ; 系統時間年月日08
D7318  ; 系統時間年月日09
D7319  ; 系統時間年月日09
D7320  ; 系統時間年月日10
D7321  ; 系統時間年月日10
D7322  ; 系統時間年月日11
D7323  ; 系統時間年月日11
D7324  ; 系統時間年月日12
D7325  ; 系統時間年月日12
D7326  ; 系統時間年月日13
D7327  ; 系統時間年月日13
D7328  ; 系統時間年月日14
D7329  ; 系統時間年月日14
D7330  ; 系統時間年月日15
D7331  ; 系統時間年月日15
D7332  ; 系統時間年月日16
D7333  ; 系統時間年月日16
D7334  ; 系統時間年月日17
D7335  ; 系統時間年月日17
D7336  ; 系統時間年月日18
D7337  ; 系統時間年月日18
D7338  ; 系統時間年月日19
D7339  ; 系統時間年月日19
D7340  ; 系統時間年月日20
D7341  ; 系統時間年月日20
D7342  ; 系統時間年月日21
D7343  ; 系統時間年月日21
D7344  ; 系統時間年月日22
D7345  ; 系統時間年月日22
D7346  ; 系統時間年月日23
D7347  ; 系統時間年月日23
D7348  ; 系統時間年月日24
D7349  ; 系統時間年月日24
D7402  ; 現在時間時分02
D7403  ; 現在時間時分03
D7404  ; 現在時間時分04
D7405  ; 現在時間時分05
D7406  ; 現在時間時分06
D7407  ; 現在時間時分07
D7408  ; 現在時間時分08
D7409  ; 現在時間時分09
D7410  ; 現在時間時分10
D7411  ; 現在時間時分11
D7412  ; 現在時間時分12
D7413  ; 現在時間時分13
D7414  ; 現在時間時分14
D7415  ; 現在時間時分15
D7416  ; 現在時間時分16
D7417  ; 現在時間時分17
D7418  ; 現在時間時分18
D7419  ; 現在時間時分19
D7420  ; 現在時間時分20
D7421  ; 現在時間時分21
D7422  ; 現在時間時分22
D7423  ; 現在時間時分23
D7424  ; 現在時間時分24
D7503  ; 本班產量履歷01
D7504  ; 本班產量履歷02
D7505  ; 本班產量履歷02
D7506  ; 本班產量履歷03
D7507  ; 本班產量履歷03
D7508  ; 本班產量履歷04
D7509  ; 本班產量履歷04
D7510  ; 本班產量履歷05
D7511  ; 本班產量履歷05
D7512  ; 本班產量履歷06
D7513  ; 本班產量履歷06
D7514  ; 本班產量履歷07
D7515  ; 本班產量履歷07
D7516  ; 本班產量履歷08
D7517  ; 本班產量履歷08
D7518  ; 本班產量履歷09
D7519  ; 本班產量履歷09
D7520  ; 本班產量履歷10
D7521  ; 本班產量履歷10
D7522  ; 本班產量履歷11
D7523  ; 本班產量履歷11
D7524  ; 本班產量履歷12
D7525  ; 本班產量履歷12
D7526  ; 本班產量履歷13
D7527  ; 本班產量履歷13
D7528  ; 本班產量履歷14
D7529  ; 本班產量履歷14
D7530  ; 本班產量履歷15
D7531  ; 本班產量履歷15
D7532  ; 本班產量履歷16
D7533  ; 本班產量履歷16
D7534  ; 本班產量履歷17
D7535  ; 本班產量履歷17
D7536  ; 本班產量履歷18
D7537  ; 本班產量履歷18
D7538  ; 本班產量履歷19
D7539  ; 本班產量履歷19
D7540  ; 本班產量履歷20
D7541  ; 本班產量履歷20
D7542  ; 本班產量履歷21
D7543  ; 本班產量履歷21
D7544  ; 本班產量履歷22
D7545  ; 本班產量履歷22
D7546  ; 本班產量履歷23
D7547  ; 本班產量履歷23
D7548  ; 本班產量履歷24
D7549  ; 本班產量履歷24
D7691  ; Buffer 2
D7693  ; Buffer 4
D10364  ; 電流PV
D10536  ; SECS_上位傳PP_SEL-QTY(ASC)
D10537  ; SECS_上位傳PP_SEL-QTY(ASC)
D10661  ; SECS_上位下PAUSE指令
D10662  ; SECS_上位下PAUSE指令
D11100  ; PV電熱01
D11102  ; PV電熱02
D11104  ; PV電熱03
D11106  ; PV電熱04
D11108  ; PV電熱05
D11110  ; PV電熱06
D11112  ; PV電熱07
D11114  ; PV電熱08
D11116  ; PV電熱09
D11118  ; PV電熱10
D11120  ; PV電熱11
D11122  ; PV電熱12
D11172  ; SV電熱01
D11174  ; SV電熱02
D11176  ; SV電熱03
D11178  ; SV電熱04
D11180  ; SV電熱05
D11182  ; SV電熱06
D11184  ; SV電熱07
D11186  ; SV電熱08
D11188  ; SV電熱09
D11190  ; SV電熱10
D11192  ; SV電熱11
D11194  ; SV電熱12
D11244  ; 左IR輸送速度設定值
D11245  ; 左IR輸送速度設定值
D11246  ; 右IR輸送速度設定值
D11247  ; 右IR輸送速度設定值
D11248  ; 上游給板尺寸寬
D11249  ; 上游給板尺寸寬
D11250  ; 上游給板尺寸長
D11251  ; 上游給板尺寸長
D12012  ; PV H13
D12013  ; PV H14
D12014  ; PV H15
D12015  ; PV H16
D12016  ; PV H17
D12017  ; PV H18
D12018  ; PV H19
D12019  ; PV H20
D12026  ; SV IRA01_FLT
D12030  ; SV H01_FLT
D12072  ; PV IRA13
D12073  ; PV IRA14
D12074  ; PV IRA15
D12075  ; PV IRA16
D12076  ; PV IRA17
D12077  ; PV IRA18
D12078  ; PV IRA19
D12079  ; PV IRA20
D12090  ; SV IRA01_FLT
D12132  ; PV IRB13
D12133  ; PV IRB14
D12134  ; PV IRB15
D12135  ; PV IRB16
D12136  ; PV IRB17
D12137  ; PV IRB18
D12138  ; PV IRB19
D12139  ; PV IRB20
D12192  ; SV H13
D12193  ; SV H14
D12194  ; SV H15
D12195  ; SV H16
D12196  ; SV H17
D12197  ; SV H18
D12198  ; SV H19
D12199  ; SV H20
D12252  ; SV IRA13
D12253  ; SV IRA14
D12254  ; SV IRA15
D12255  ; SV IRA16
D12256  ; SV IRA17
D12257  ; SV IRA18
D12258  ; SV IRA19
D12259  ; SV IRA20
D12312  ; SV IRB13
D12313  ; SV IRB14
D12314  ; SV IRB15
D12315  ; SV IRB16
D12316  ; SV IRB17
D12317  ; SV IRB18
D12318  ; SV IRB19
D12319  ; SV IRB20
D12364  ; 電流PV
D13100  ; BF-SV H01
D13601  ; 配方設定SV H02
D13602  ; 配方設定SV H03
D13603  ; 配方設定SV H04
D13604  ; 配方設定SV H05
D13605  ; 配方設定SV H06
D13606  ; 配方設定SV H07
D13607  ; 配方設定SV H08
D13608  ; 配方設定SV H09
D13609  ; 配方設定SV H10
D13610  ; 配方設定SV H11
D13611  ; 配方設定SV H12
D13620  ; 配方設定SV IRA01
D13621  ; 配方設定SV IRA02
D13622  ; 配方設定SV IRA03
D13623  ; 配方設定SV IRA04
D13624  ; 配方設定SV IRA05
D13625  ; 配方設定SV IRA06
D13626  ; 配方設定SV IRA07
D13627  ; 配方設定SV IRA08
D13628  ; 配方設定SV IRA09
D13629  ; 配方設定SV IRA10
D13630  ; 配方設定SV IRA11
D13631  ; 配方設定SV IRA12
D13640  ; 配方設定SV IRB01
D13641  ; 配方設定SV IRB02
D13642  ; 配方設定SV IRB03
D13643  ; 配方設定SV IRB04
D13644  ; 配方設定SV IRB05
D13645  ; 配方設定SV IRB06
D13646  ; 配方設定SV IRB07
D13647  ; 配方設定SV IRB08
D13648  ; 配方設定SV IRB09
D13649  ; 配方設定SV IRB10
D13650  ; 配方設定SV IRB11
D13651  ; 配方設定SV IRB12
D13660  ; 配方設定輸送速度左IR
D13661  ; 配方設定輸送速度右IR
D14550  ; QTY數量
D20202  ; C1
D20203  ; D1
D20204  ; E1
D20205  ; F1
D20206  ; G1
D20207  ; H1
D20208  ; I1
D20209  ; J1
D22540  ; SECS-上傳新增刪除修改名稱
D24550  ; QTY數量
D25340  ; A
D25341  ; B
D25342  ; C
D25343  ; D
D25344  ; E
D25345  ; F
D25346  ; G
D25347  ; H
D25348  ; I
D25349  ; J
D25350  ; K
D25351  ; L
D25352  ; M
D25353  ; N
D25354  ; O
D25355  ; P
D25356  ; Q
D25357  ; R
D25358  ; S
D25359  ; T
D25379  ; SECS暫存判斷寫入電熱1-SV用
D25409  ; 配方組別
D25413  ; HMI-編輯烘烤步進時間設定
D25512  ; 配方組別計算暫存
D25513  ; 配方組別計算-1(-1)
D25515  ; 配方組別計算
D26390  ; S-BF
D26400  ; S-選擇配方名稱BF
P10  ; 手動加熱狀態
P2000  ; SPARE
P3000  ; 出料手臂ROBOT
ZR0  ; 密碼權限設定01
ZR1  ; 密碼權限設定01
ZR2  ; 密碼權限設定02
ZR3  ; 密碼權限設定02
ZR5  ; 密碼權限設定03
ZR6  ; 密碼權限設定04
ZR7  ; 密碼權限設定04
ZR8  ; 密碼權限設定05
ZR9  ; 密碼權限設定05
ZR10  ; 密碼權限設定06
ZR11  ; 密碼權限設定06
ZR12  ; 密碼權限設定07
ZR13  ; 密碼權限設定07
ZR14  ; 密碼權限設定08
ZR15  ; 密碼權限設定08
ZR16  ; 密碼權限設定09
ZR17  ; 密碼權限設定09
ZR18  ; 密碼權限設定10
ZR19  ; 密碼權限設定10
ZR20  ; 密碼權限設定11
ZR21  ; 密碼權限設定11
ZR22  ; 密碼權限設定12
ZR23  ; 密碼權限設定12
ZR24  ; 密碼權限設定13
ZR25  ; 密碼權限設定13
ZR26  ; 密碼權限設定14
ZR27  ; 密碼權限設定14
ZR28  ; 密碼權限設定15
ZR29  ; 密碼權限設定15
ZR1101  ; 整板寸動設定速度
ZR1105  ; 整板現在位置Range_+
ZR1107  ; 整板現在位置Range_-
ZR1111  ; 整板速度01
ZR1113  ; 整板位置01
ZR1121  ; 整板速度02
ZR1123  ; 整板位置02
ZR1131  ; 整板速度03
ZR1133  ; 整板位置03
ZR1140  ; 整板速度04
ZR1141  ; 整板速度04
ZR1143  ; 整板位置04
ZR1150  ; 整板速度05
ZR1151  ; 整板速度05
ZR1152  ; 整板位置05
ZR1153  ; 整板位置05
ZR1160  ; 整板速度06
ZR1161  ; 整板速度06
ZR1162  ; 整板位置06
ZR1163  ; 整板位置06
ZR1170  ; 整板速度07
ZR1171  ; 整板速度07
ZR1172  ; 整板位置07
ZR1173  ; 整板位置07
ZR1180  ; 整板速度08
ZR1181  ; 整板速度08
ZR1182  ; 整板位置08
ZR1183  ; 整板位置08
ZR1190  ; 整板速度09
ZR1191  ; 整板速度09
ZR1192  ; 整板位置09
ZR1193  ; 整板位置09
ZR1201  ; 牙插移載寸動設定速度
ZR1205  ; 牙插移載現在位置Range_+
ZR1207  ; 牙插移載現在位置Range_-
ZR1211  ; 牙插移載速度01
ZR1213  ; 牙插移載位置01
ZR1221  ; 牙插移載速度02
ZR1223  ; 牙插移載位置02
ZR1230  ; 牙插移載速度03
ZR1231  ; 牙插移載速度03
ZR1233  ; 牙插移載位置03
ZR1240  ; 牙插移載速度04
ZR1241  ; 牙插移載速度04
ZR1243  ; 牙插移載位置04
ZR1250  ; 牙插移載速度05
ZR1251  ; 牙插移載速度05
ZR1260  ; 牙插移載速度06
ZR1261  ; 牙插移載速度06
ZR1270  ; 牙插移載速度07
ZR1271  ; 牙插移載速度07
ZR1280  ; 牙插移載速度08
ZR1281  ; 牙插移載速度08
ZR1290  ; 牙插移載速度09
ZR1291  ; 牙插移載速度09
ZR1401  ; 進手臂取手寸動設定速度
ZR1405  ; 進手臂取手現在位置Range_+
ZR1407  ; 進手臂取手現在位置Range_-
ZR1411  ; 進手臂取手速度01
ZR1413  ; 進手臂取手位置01
ZR1421  ; 進手臂取手速度02
ZR1423  ; 進手臂取手位置02
ZR1430  ; 進手臂取手速度03
ZR1431  ; 進手臂取手速度03
ZR1433  ; 進手臂取手位置03
ZR1440  ; 進手臂取手速度04
ZR1441  ; 進手臂取手速度04
ZR1443  ; 進手臂取手位置04
ZR1450  ; 進手臂取手速度05
ZR1451  ; 進手臂取手速度05
ZR1460  ; 進手臂取手速度06
ZR1461  ; 進手臂取手速度06
ZR1470  ; 進手臂取手速度07
ZR1471  ; 進手臂取手速度07
ZR1480  ; 進手臂取手速度08
ZR1481  ; 進手臂取手速度08
ZR1490  ; 進手臂取手速度09
ZR1491  ; 進手臂取手速度09
ZR1501  ; 進料托框昇降寸動設定速度
ZR1505  ; 進料托框昇降現在位置Range_+
ZR1507  ; 進料托框昇降現在位置Range_-
ZR1511  ; 進料托框昇降速度01
ZR1513  ; 進料托框昇降位置01
ZR1521  ; 進料托框昇降速度02
ZR1523  ; 進料托框昇降位置02
ZR1531  ; 進料托框昇降速度03
ZR1533  ; 進料托框昇降位置03
ZR1541  ; 進料托框昇降速度04
ZR1543  ; 進料托框昇降位置04
ZR1550  ; 進料托框昇降速度05
ZR1551  ; 進料托框昇降速度05
ZR1552  ; 進料托框昇降位置05
ZR1553  ; 進料托框昇降位置05
ZR1560  ; 進料托框昇降速度06
ZR1561  ; 進料托框昇降速度06
ZR1570  ; 進料托框昇降速度07
ZR1571  ; 進料托框昇降速度07
ZR1580  ; 進料托框昇降速度08
ZR1581  ; 進料托框昇降速度08
ZR1590  ; 進料托框昇降速度09
ZR1591  ; 進料托框昇降速度09
ZR1592  ; 進料托框昇降位置09
ZR1593  ; 進料托框昇降位置09
ZR1601  ; 進左開爪寸動設定速度
ZR1605  ; 進左開爪現在位置Range_+
ZR1607  ; 進左開爪現在位置Range_-
ZR1611  ; 進左開爪速度01
ZR1613  ; 進左開爪位置01
ZR1621  ; 進左開爪速度02
ZR1623  ; 進左開爪位置02
ZR1631  ; 進左開爪速度03
ZR1633  ; 進左開爪位置03
ZR1641  ; 進左開爪速度04
ZR1643  ; 進左開爪位置04
ZR1651  ; 進左開爪速度05
ZR1653  ; 進左開爪位置05
ZR1660  ; 進左開爪速度06
ZR1661  ; 進左開爪速度06
ZR1670  ; 進左開爪速度07
ZR1671  ; 進左開爪速度07
ZR1680  ; 進左開爪速度08
ZR1681  ; 進左開爪速度08
ZR1690  ; 進左開爪速度09
ZR1691  ; 進左開爪速度09
ZR1701  ; 進右開爪寸動設定速度
ZR1705  ; 進右開爪現在位置Range_+
ZR1707  ; 進右開爪現在位置Range_-
ZR1711  ; 進右開爪速度01
ZR1713  ; 進右開爪位置01
ZR1721  ; 進右開爪速度02
ZR1723  ; 進右開爪位置02
ZR1731  ; 進右開爪速度03
ZR1733  ; 進右開爪位置03
ZR1741  ; 進右開爪速度04
ZR1743  ; 進右開爪位置04
ZR1751  ; 進右開爪速度05
ZR1753  ; 進右開爪位置05
ZR1760  ; 進右開爪速度06
ZR1761  ; 進右開爪速度06
ZR1770  ; 進右開爪速度07
ZR1771  ; 進右開爪速度07
ZR1780  ; 進右開爪速度08
ZR1781  ; 進右開爪速度08
ZR1790  ; 進右開爪速度09
ZR1791  ; 進右開爪速度09
ZR2010  ; 烘烤時間設定MIN
ZR2012  ; 烘烤時間設定SEC
ZR2013  ; 烘烤時間設定SEC
ZR2020  ; 烘烤時間設定MIN 暫存
ZR2022  ; 烘烤時間設定SEC 暫存
ZR2024  ; 烘烤步進間隔時間SEC BF
ZR2029  ; 配方內容組數
ZR2030  ; 加熱段  總框架數
ZR2032  ; 爐體冷卻總框架數
ZR2036  ; 烘烤時間設定    總秒數
ZR2038  ; 烘烤步進間隔時間SEC
ZR2101  ; 分流前取框寸動設定速度
ZR2105  ; 分流前取框現在位置Range_+
ZR2107  ; 分流前取框現在位置Range_-
ZR2111  ; 分流前取框速度01
ZR2113  ; 分流前取框位置01
ZR2121  ; 分流前取框速度02
ZR2123  ; 分流前取框位置02
ZR2131  ; 分流前取框速度03
ZR2133  ; 分流前取框位置03
ZR2140  ; 分流前取框速度04
ZR2141  ; 分流前取框速度04
ZR2143  ; 分流前取框位置04
ZR2150  ; 分流前取框速度05
ZR2151  ; 分流前取框速度05
ZR2160  ; 分流前取框速度06
ZR2161  ; 分流前取框速度06
ZR2170  ; 分流前取框速度07
ZR2171  ; 分流前取框速度07
ZR2180  ; 分流前取框速度08
ZR2181  ; 分流前取框速度08
ZR2190  ; 分流前取框速度09
ZR2191  ; 分流前取框速度09
ZR2201  ; 合流後掛框寸動設定速度
ZR2203  ; 合流後掛框Servo   Intrval Pitch
ZR2205  ; 合流後掛框現在位置Range_+
ZR2207  ; 合流後掛框現在位置Range_-
ZR2211  ; 合流後掛框速度01
ZR2213  ; 合流後掛框位置01
ZR2221  ; 合流後掛框速度02
ZR2223  ; 合流後掛框位置02
ZR2231  ; 合流後掛框速度03
ZR2233  ; 合流後掛框位置03
ZR2240  ; 合流後掛框速度04
ZR2241  ; 合流後掛框速度04
ZR2243  ; 合流後掛框位置04
ZR2250  ; 合流後掛框速度05
ZR2251  ; 合流後掛框速度05
ZR2260  ; 合流後掛框速度06
ZR2261  ; 合流後掛框速度06
ZR2270  ; 合流後掛框速度07
ZR2271  ; 合流後掛框速度07
ZR2280  ; 合流後掛框速度08
ZR2281  ; 合流後掛框速度08
ZR2290  ; 合流後掛框速度09
ZR2291  ; 合流後掛框速度09
ZR3101  ; 出手臂取手寸動設定速度
ZR3103  ; 出手臂取手Servo   Intrval Pitch
ZR3105  ; 出手臂取手現在位置Range_+
ZR3107  ; 出手臂取手現在位置Range_-
ZR3111  ; 出手臂取手速度01
ZR3113  ; 出手臂取手位置01
ZR3121  ; 出手臂取手速度02
ZR3123  ; 出手臂取手位置02
ZR3131  ; 出手臂取手速度03
ZR3133  ; 出手臂取手位置03
ZR3140  ; 出手臂取手速度04
ZR3141  ; 出手臂取手速度04
ZR3143  ; 出手臂取手位置04
ZR3150  ; 出手臂取手速度05
ZR3151  ; 出手臂取手速度05
ZR3160  ; 出手臂取手速度06
ZR3161  ; 出手臂取手速度06
ZR3170  ; 出手臂取手速度07
ZR3171  ; 出手臂取手速度07
ZR3180  ; 出手臂取手速度08
ZR3181  ; 出手臂取手速度08
ZR3190  ; 出手臂取手速度09
ZR3191  ; 出手臂取手速度09
ZR3201  ; 出料托框昇降寸動設定速度
ZR3203  ; 出料托框昇降Servo   Intrval Pitc
ZR3205  ; 出料托框昇降現在位置Range_+
ZR3207  ; 出料托框昇降現在位置Range_-
ZR3211  ; 出料托框昇降速度01
ZR3213  ; 出料托框昇降位置01
ZR3221  ; 出料托框昇降速度02
ZR3223  ; 出料托框昇降位置02
ZR3231  ; 出料托框昇降速度03
ZR3233  ; 出料托框昇降位置03
ZR3241  ; 出料托框昇降速度04
ZR3243  ; 出料托框昇降位置04
ZR3251  ; 出料托框昇降速度05
ZR3253  ; 出料托框昇降位置05
ZR3260  ; 出料托框昇降速度06
ZR3261  ; 出料托框昇降速度06
ZR3270  ; 出料托框昇降速度07
ZR3271  ; 出料托框昇降速度07
ZR3280  ; 出料托框昇降速度08
ZR3281  ; 出料托框昇降速度08
ZR3290  ; 出料托框昇降速度09
ZR3291  ; 出料托框昇降速度09
ZR3292  ; 出料托框昇降位置09
ZR3293  ; 出料托框昇降位置09
ZR3301  ; 出左開夾寸動設定速度
ZR3303  ; 出左開夾Servo   Intrval Pitch
ZR3305  ; 出左開夾現在位置Range_+
ZR3307  ; 出左開夾現在位置Range_-
ZR3311  ; 出左開夾速度01
ZR3313  ; 出左開夾位置01
ZR3321  ; 出左開夾速度02
ZR3323  ; 出左開夾位置02
ZR3331  ; 出左開夾速度03
ZR3333  ; 出左開夾位置03
ZR3341  ; 出左開夾速度04
ZR3343  ; 出左開夾位置04
ZR3351  ; 出左開夾速度05
ZR3353  ; 出左開夾位置05
ZR3360  ; 出左開夾速度06
ZR3361  ; 出左開夾速度06
ZR3370  ; 出左開夾速度07
ZR3371  ; 出左開夾速度07
ZR3380  ; 出左開夾速度08
ZR3381  ; 出左開夾速度08
ZR3390  ; 出左開夾速度09
ZR3391  ; 出左開夾速度09
ZR3401  ; 出右開夾寸動設定速度
ZR3403  ; 出右開夾Servo   Intrval Pitch
ZR3405  ; 出右開夾現在位置Range_+
ZR3407  ; 出右開夾現在位置Range_-
ZR3411  ; 出右開夾速度01
ZR3413  ; 出右開夾位置01
ZR3421  ; 出右開夾速度02
ZR3423  ; 出右開夾位置02
ZR3431  ; 出右開夾速度03
ZR3433  ; 出右開夾位置03
ZR3441  ; 出右開夾速度04
ZR3443  ; 出右開夾位置04
ZR3451  ; 出右開夾速度05
ZR3453  ; 出右開夾位置05
ZR3460  ; 出右開夾速度06
ZR3461  ; 出右開夾速度06
ZR3470  ; 出右開夾速度07
ZR3471  ; 出右開夾速度07
ZR3480  ; 出右開夾速度08
ZR3481  ; 出右開夾速度08
ZR3490  ; 出右開夾速度09
ZR3491  ; 出右開夾速度09
ZR3501  ; 出板牙插移載寸動設定速度
ZR3505  ; 出板牙插移載現在位置Range_+
ZR3507  ; 出板牙插移載現在位置Range_-
ZR3511  ; 出板牙插移載速度01
ZR3513  ; 出板牙插移載位置01
ZR3521  ; 出板牙插移載速度02
ZR3523  ; 出板牙插移載位置02
ZR3531  ; 出板牙插移載速度03
ZR3533  ; 出板牙插移載位置03
ZR3540  ; 出板牙插移載速度04
ZR3541  ; 出板牙插移載速度04
ZR3543  ; 出板牙插移載位置04
ZR3550  ; 出板牙插移載速度05
ZR3551  ; 出板牙插移載速度05
ZR3560  ; 出板牙插移載速度06
ZR3561  ; 出板牙插移載速度06
ZR3570  ; 出板牙插移載速度07
ZR3571  ; 出板牙插移載速度07
ZR3580  ; 出板牙插移載速度08
ZR3581  ; 出板牙插移載速度08
ZR3590  ; 出板牙插移載速度09
ZR3591  ; 出板牙插移載速度09
ZR5000  ; HMI-溫度配方 電熱1-SV
ZR5029  ; 配方組別
ZR5200  ; SECS_上位配方_1使用/0不使用
ZR5201  ; SECS_上位配方NO.01
ZR5300  ; 所有設定配方名稱1
ZR5302  ; PPID(Name)
ZR10000  ; 配風設定內容BF第一個word
ZR31000  ; 配方組別bf
B2E  ; 連線上游備用
B2F  ; 連線上游備用
B0FE  ; 電源相序檢知
B120  ; 第01槽風車馬達過載異常
B121  ; 第02槽風車馬達過載異常
B122  ; 第03槽風車馬達過載異常
B123  ; 第04槽風車馬達過載異常
B124  ; 第05槽風車馬達過載異常
B125  ; 第06槽風車馬達過載異常
B126  ; 第07槽風車馬達過載異常
B127  ; 第08槽風車馬達過載異常
B128  ; 第01槽風車馬達電流檢知
B129  ; 第02槽風車馬達電流檢知
B12A  ; 第03槽風車馬達電流檢知
B12B  ; 第04槽風車馬達電流檢知
B12C  ; 第05槽風車馬達電流檢知
B12D  ; 第06槽風車馬達電流檢知
B12E  ; 第07槽風車馬達電流檢知
B12F  ; 第08槽風車馬達電流檢知
B130  ; 第01槽電熱箱H01超溫防止器
B131  ; 第02槽電熱箱H02超溫防止器
B132  ; 第03槽電熱箱H03超溫防止器
B133  ; 第04槽電熱箱H04超溫防止器
B134  ; 第05槽電熱箱H05超溫防止器
B135  ; 第06槽電熱箱H06超溫防止器
B136  ; 第07槽電熱箱H07超溫防止器
B137  ; 第08槽電熱箱H08超溫防止器
B138  ; 第01槽IR01A超溫防止器
B139  ; 第02槽IR02A超溫防止器
B13A  ; 第03槽IR03A超溫防止器
B13B  ; 第04槽IR04A超溫防止器
B13C  ; 第05槽IR05A超溫防止器
B13D  ; 第06槽IR06A超溫防止器
B13E  ; 第07槽IR07A超溫防止器
B13F  ; 第08槽IR08A超溫防止器
B140  ; 第01槽熱風H01溫度到達
B141  ; 第02槽熱風H02溫度到達
B142  ; 第03槽熱風H03溫度到達
B143  ; 第04槽熱風H04溫度到達
B144  ; 第05槽熱風H05溫度到達
B145  ; 第06槽熱風H06溫度到達
B146  ; 第07槽熱風H07溫度到達
B147  ; 第08槽熱風H08溫度到達
B148  ; 第01槽IR01A溫度到達
B149  ; 第02槽IR02A溫度到達
B14A  ; 第03槽IR03A溫度到達
B14B  ; 第04槽IR04A溫度到達
B14C  ; 第05槽IR05A溫度到達
B14D  ; 第06槽IR06A溫度到達
B14E  ; 第07槽IR07A溫度到達
B14F  ; 第08槽IR08A溫度到達
B150  ; 第01槽H01溫控超溫異常
B151  ; 第02槽H02溫控超溫異常
B152  ; 第03槽H03溫控超溫異常
B153  ; 第04槽H04溫控超溫異常
B154  ; 第05槽H05溫控超溫異常
B155  ; 第06槽H06溫控超溫異常
B156  ; 第07槽H07溫控超溫異常
B157  ; 第08槽H08溫控超溫異常
B158  ; 第01槽IR01A溫控超溫異常
B159  ; 第02槽IR02A溫控超溫異常
B15A  ; 第03槽IR03A溫控超溫異常
B15B  ; 第04槽IR04A溫控超溫異常
B15C  ; 第05槽IR05A溫控超溫異常
B15D  ; 第06槽IR06A溫控超溫異常
B15E  ; 第07槽IR07A溫控超溫異常
B15F  ; 第08槽IR08A溫控超溫異常
B168  ; 第09槽SCR09/09A/09B異常
B169  ; 第10槽SCR10/10A/10B異常
B16A  ; 第11槽SCR11/911/11B異常
B16B  ; 第12槽SCR12/12A/12B異常
B16C  ; 第09槽分路開關跳脫異常
B16D  ; 第10槽分路開關跳脫異常
B170  ; 第01槽SCR01/01A/01B異常
B171  ; 第02槽SCR02/02A/02B異常
B172  ; 第03槽SCR03/03A/03B異常
B173  ; 第04槽SCR04/04A/04B異常
B174  ; 第05槽SCR05/05A/05B異常
B175  ; 第06槽SCR06/06A/06B異常
B176  ; 第07槽SCR07/07A/07B異常
B177  ; 第08槽SCR08/08A/08B異常
B178  ; 第01槽分路開關跳脫異常
B179  ; 第02槽分路開關跳脫異常
B17A  ; 第03槽分路開關跳脫異常
B17B  ; 第04槽分路開關跳脫異常
B17C  ; 第05槽分路開關跳脫異常
B17D  ; 第06槽分路開關跳脫異常
B17E  ; 第07槽分路開關跳脫異常
B17F  ; 第08槽分路開關跳脫異常
B180  ; 第01槽IR01B溫度到達
B181  ; 第02槽IR02B溫度到達
B182  ; 第03槽IR03B溫度到達
B183  ; 第04槽IR04B溫度到達
B184  ; 第05槽IR05B溫度到達
B185  ; 第06槽IR06B溫度到達
B186  ; 第07槽IR07B溫度到達
B187  ; 第08槽IR08B溫度到達
B188  ; 第01槽IR01B超溫防止器
B189  ; 第02槽IR02B超溫防止器
B18A  ; 第03槽IR03B超溫防止器
B18B  ; 第04槽IR04B超溫防止器
B18C  ; 第05槽IR05B超溫防止器
B18D  ; 第06槽IR06B超溫防止器
B18E  ; 第07槽IR07B超溫防止器
B18F  ; 第08槽IR08B超溫防止器
B190  ; 第01槽IR01B溫控超溫異常
B191  ; 第02槽IR02B溫控超溫異常
B192  ; 第03槽IR03B溫控超溫異常
B193  ; 第04槽IR04B溫控超溫異常
B194  ; 第05槽IR05B溫控超溫異常
B195  ; 第06槽IR06B溫控超溫異常
B196  ; 第07槽IR07B溫控超溫異常
B197  ; 第08槽IR08B溫控超溫異常
B1A0  ; 第09槽熱風H09溫度到達
B1A2  ; 第09槽IR09A溫度到達
B1A4  ; 第09槽IR09B溫度到達
B1A8  ; 第10槽熱風H10溫度到達
B1AA  ; 第10槽IR10A溫度到達
B1AC  ; 第10槽IR10B溫度到達
B1B0  ; 第11槽熱風H11溫度到達
B1B2  ; 第11槽IR11A溫度到達
B1B4  ; 第11槽IR11B溫度到達
B1B8  ; 第12槽熱風H12溫度到達
B1B9  ; 第12槽H12溫控超溫異常
B1BA  ; 第12槽IR12A溫度到達
B1BC  ; 第12槽IR12B溫度到達
B1BE  ; 第11槽風車變頻機INV11運轉
B1BF  ; 第12槽風車變頻機INV12運轉
B21E  ; CCD照明繼電器
B26F  ; 出料變頻器異常復歸
B28E  ; 出料輸送變頻器INVC2慢速
B2BC  ; 進料輸送排氣電磁開關
B2BD  ; 出料輸送排氣電磁開關
B501  ; 第02槽  熱風電磁開關
B502  ; 第03槽  熱風電磁開關
B503  ; 第04槽  熱風電磁開關
B504  ; 第05槽  熱風電磁開關
B505  ; 第06槽  熱風電磁開關
B506  ; 第07槽  熱風電磁開關
B507  ; 第08槽  熱風電磁開關
B508  ; 第09槽  熱風電磁開關
B509  ; 第10槽  熱風電磁開關
B50A  ; 第11槽  熱風電磁開關
B50B  ; 第12槽  熱風電磁開關
B50C  ; 第13槽  熱風電磁開關
B50D  ; 第14槽  熱風電磁開關
B50E  ; 第15槽  熱風電磁開關
B50F  ; 第16槽  熱風電磁開關
B511  ; 第02槽  IRA 電磁開關
B512  ; 第03槽  IRA 電磁開關
B513  ; 第04槽  IRA 電磁開關
B514  ; 第05槽  IRA 電磁開關
B515  ; 第06槽  IRA 電磁開關
B516  ; 第07槽  IRA 電磁開關
B517  ; 第08槽  IRA 電磁開關
B518  ; 第09槽  IRA 電磁開關
B519  ; 第10槽  IRA 電磁開關
B51A  ; 第11槽  IRA 電磁開關
B51B  ; 第12槽  IRA 電磁開關
B51C  ; 第13槽  IRA 電磁開關
B51D  ; 第14槽  IRA 電磁開關
B51E  ; 第15槽  IRA 電磁開關
B51F  ; 第16槽  IRA 電磁開關
B521  ; 第02槽  IRB 電磁開關
B522  ; 第03槽  IRB 電磁開關
B523  ; 第04槽  IRB 電磁開關
B524  ; 第05槽  IRB 電磁開關
B525  ; 第06槽  IRB 電磁開關
B526  ; 第07槽  IRB 電磁開關
B527  ; 第08槽  IRB 電磁開關
B528  ; 第09槽  IRB 電磁開關
B529  ; 第10槽  IRB 電磁開關
B52A  ; 第11槽  IRB 電磁開關
B52B  ; 第12槽  IRB 電磁開關
B52C  ; 第13槽  IRB 電磁開關
B52D  ; 第14槽  IRB 電磁開關
B52E  ; 第15槽  IRB 電磁開關
B52F  ; 第16槽  IRB 電磁開關
B804  ; 掉框板異常
B80A  ; 低溫異常數量
B80B  ; ELB 跳脫異常數量
B1014  ; 進料手臂下夾板  夾
B1015  ; 進料手臂下夾板  放
B110A  ; 重要異常
B110B  ; EGO 超溫異常數量
B1200  ; 爐體重要異常警報
B1202  ; 風車異常警報
B1203  ; 超溫異常警報
B1204  ; 低溫異常警報
B1205  ; 昇降搬移異常警報
B1206  ; 爐體異常警告
B1207  ; 爐體段保養時間到達警報
B1208  ; ELB 跳脫異常
B120A  ; 爐體SEN 異常
B1221  ; 進料牙插移載允許位置01
B1222  ; 進料牙插移載允許位置02
B1223  ; 進料牙插移載允許位置03
B1224  ; 進料牙插移載允許位置04
B1300  ; 出料重要異常
B1421  ; 進料手臂取手允許位置01
B1422  ; 進料手臂取手允許位置02
B1423  ; 進料手臂取手允許位置03
B1424  ; 進料手臂取手允許位置04
B1621  ; 進左開爪允許位置01
B1622  ; 進左開爪允許位置02
B1623  ; 進左開爪允許位置03
B1624  ; 進左開爪允許位置04
B1721  ; 進右開爪允許位置01
B1722  ; 進右開爪允許位置02
B1723  ; 進右開爪允許位置03
B1724  ; 進右開爪允許位置04
B2124  ; 進料分流取框允許位置04
B2223  ; 出料合流取框允許位置03
B2224  ; 出料合流取框允許位置03
B30E0  ; 停止PLS
B30E1  ; 加熱01  停止PLS
B30E2  ; 加熱02  停止PLS
B30E3  ; 加熱03  停止PLS
B30E4  ; 加熱04  停止PLS
B30E5  ; 加熱05  停止PLS
B30E6  ; 加熱06  停止PLS
B30E7  ; 加熱07  停止PLS
B30E8  ; 加熱08  停止PLS
B30E9  ; 加熱09  停止PLS
B30EA  ; 加熱10  停止PLS
B30EB  ; 加熱11  停止PLS
B30EC  ; 加熱12  停止PLS
B30ED  ; 循環風車01停止PLS
B30EE  ; 循環風車02停止PLS
B30EF  ; 循環風車03停止PLS
B30F0  ; 循環風車04停止PLS
B30F1  ; 循環風車05停止PLS
B30F2  ; 循環風車06停止PLS
B30F3  ; 循環風車07停止PLS
B30F4  ; 循環風車08停止PLS
B30F5  ; 循環風車09停止PLS
B30F6  ; 循環風車10停止PLS
B30F7  ; 循環風車11停止PLS
B30F8  ; 循環風車12停止PLS
B30F9  ; 進料排氣風車停止PLS
B30FA  ; 出料冷卻1風車停止PLS
B30FB  ; 出料冷卻2風車停止PLS
B3121  ; 出料手臂取手允許位置01
B3122  ; 出料手臂取手允許位置02
B3123  ; 出料手臂取手允許位置03
B3124  ; 出料手臂取手允許位置04
B3157  ; 進料機構原點停止
B3221  ; 出料托框昇降允許位置01
B3222  ; 出料托框昇降允許位置02
B3223  ; 出料托框昇降允許位置03
B3224  ; 出料托框昇降允許位置04
B323D  ; 出料輸送再啟動信號
B3321  ; 出料左側開爪允許位置01
B3322  ; 出料左側開爪允許位置02
B3323  ; 出料左側開爪允許位置03
B3324  ; 出料左側開爪允許位置04
B3325  ; 出料左側開爪允許位置05
B3341  ; 進料安全門警報不停機
B3343  ; 進料電動門不使用
B3351  ; 出料安全門警報不停機
B3353  ; 出料電動門不使用
B3421  ; 出料右側開爪允許位置01
B3422  ; 出料右側開爪允許位置02
B3423  ; 出料右側開爪允許位置03
B3424  ; 出料右側開爪允許位置04
B3425  ; 出料右側開爪允許位置05
B3521  ; 出料牙叉允許位置01
B3522  ; 出料牙叉允許位置02
B3523  ; 出料牙叉允許位置03
B3524  ; 出料牙叉允許位置04
B3525  ; 出料牙叉允許位置05
W1900  ; FR1(1)手臂X軸偏差位置_整數部分
W1901  ; FR1(2)手臂X軸偏差位置_小數部分
W1902  ; FR1(3)手臂Y軸偏差位置_整數部分
W1903  ; FR1(4)手臂Y軸偏差位置_小數部分
W1904  ; FR1(5)手臂T軸偏差位置_整數部分
W1905  ; FR1(6)手臂T軸偏差位置_小數部分
W1906  ; FR1(7)手臂X軸目前位置_整數部分
W1907  ; FR1(8)手臂X軸目前位置_小數部分
W1908  ; FR1(9)手臂Y軸目前位置_整數部分
W1909  ; FR1(10)手臂Y軸目前位置_小數部分
W190A  ; FR1(11)手臂T軸目前位置_整數部分
W190B  ; FR1(12)手臂T軸偏差位置_小數部分
W190C  ; FR1(13)
W190D  ; FR1(14)
W190E  ; FR1(15)
W190F  ; FR1(16)
W1910  ; FR2手臂>輸送手臂X軸偏差位置_整數
W1911  ; FR2手臂>輸送手臂X軸偏差位置_小數
W1912  ; FR2手臂>輸送手臂Y軸偏差位置_整數
W1913  ; FR2手臂>輸送手臂Y軸偏差位置_小數
W1914  ; FR2手臂>輸送手臂Z軸偏差位置_整數
W1915  ; FR2手臂>輸送手臂Z軸偏差位置_小數
W191F  ; FR2_PLCAOUT (16) = regulate_cnt
W2009  ; TR1 放板點(左右補償)Y
W200A  ; TR1 放板點(升降補償)Z
W200C  ; TR1 B(前後補償)X
W200E  ; TR1 B(升降補償)Z
W200F  ; TR1
W201B  ; TR2 L誤差/2
W201C  ; TR2 B(前後補償)X
W201D  ; TR2 w誤差/2
W201E  ; TR2 B(升降補償)Z
W201F  ; TR2
W5011  ; 出料手臂大板寬  旋轉補正整數
W5013  ; 出料手臂大板寬  旋轉補正小數
W5015  ; 出料手臂大板寬  補正整數
W5017  ; 出料手臂大板寬  補正小數
D4600.8  ; 允許啟動運轉信號8
D4600.9  ; 允許啟動運轉信號9
D4600.A  ; 允許啟動運轉信號10
D4600.B  ; 允許啟動運轉信號11
D4600.C  ; 允許啟動運轉信號12
D4600.D  ; 允許啟動運轉信號13
D4600.E  ; 允許啟動運轉信號14
D4600.F  ; 允許啟動運轉信號15
D4611.4  ; 進料牙叉原點燈_4
D4611.5  ; 進料牙叉原點燈_5
D4611.6  ; 進料牙叉原點燈_6
D4611.7  ; 進料牙叉原點燈_7
D4611.8  ; 進料牙叉原點燈_8
D4611.9  ; 進料牙叉原點燈_9
D4611.A  ; 進料牙叉原點燈_10
D4611.B  ; 進料牙叉原點燈_11
D4611.C  ; 進料牙叉原點燈_12
D4611.D  ; 進料牙叉原點燈_13
D4611.E  ; 進料牙叉原點燈_14
D4611.F  ; 進料牙叉原點燈_15
D4612.5  ; 進料手臂原點燈_5
D4612.6  ; 進料手臂原點燈_6
D4612.7  ; 進料手臂原點燈_7
D4612.8  ; 進料手臂原點燈_8
D4612.9  ; 進料手臂原點燈_9
D4612.A  ; 進料手臂原點燈_10
D4612.B  ; 進料手臂原點燈_11
D4612.C  ; 進料手臂原點燈_12
D4612.D  ; 進料手臂原點燈_13
D4612.E  ; 進料手臂原點燈_14
D4612.F  ; 進料手臂原點燈_15
D4613.5  ; 進料托框回流原點燈_5
D4613.6  ; 進料托框回流原點燈_6
D4613.7  ; 進料托框回流原點燈_7
D4613.8  ; 進料托框回流原點燈_8
D4613.9  ; 進料托框回流原點燈_9
D4613.A  ; 進料托框回流原點燈_10
D4613.B  ; 進料托框回流原點燈_11
D4613.C  ; 進料托框回流原點燈_12
D4613.D  ; 進料托框回流原點燈_13
D4613.E  ; 進料托框回流原點燈_14
D4613.F  ; 進料托框回流原點燈_15
D4614.7  ; 進料開爪原點燈_7
D4614.8  ; 進料開爪原點燈_8
D4614.9  ; 進料開爪原點燈_9
D4614.A  ; 進料開爪原點燈_10
D4614.B  ; 進料開爪原點燈_11
D4614.C  ; 進料開爪原點燈_12
D4614.D  ; 進料開爪原點燈_13
D4614.E  ; 進料開爪原點燈_14
D4614.F  ; 進料開爪原點燈_15
D4615.8  ; 進料分流原點燈_8
D4615.9  ; 進料分流原點燈_9
D4615.A  ; 進料分流原點燈_10
D4615.B  ; 進料分流原點燈_11
D4615.C  ; 進料分流原點燈_12
D4615.D  ; 進料分流原點燈_13
D4615.E  ; 進料分流原點燈_14
D4615.F  ; 進料分流原點燈_15
D4631.8  ; 出料分流原點燈_8
D4631.9  ; 出料分流原點燈_9
D4631.A  ; 出料分流原點燈_10
D4631.B  ; 出料分流原點燈_11
D4631.C  ; 出料分流原點燈_12
D4631.D  ; 出料分流原點燈_13
D4631.E  ; 出料分流原點燈_14
D4631.F  ; 出料分流原點燈_15
D4632.7  ; 出料開爪原點燈_7
D4632.8  ; 出料開爪原點燈_8
D4632.9  ; 出料開爪原點燈_9
D4632.A  ; 出料開爪原點燈_10
D4632.B  ; 出料開爪原點燈_11
D4632.C  ; 出料開爪原點燈_12
D4632.D  ; 出料開爪原點燈_13
D4632.E  ; 出料開爪原點燈_14
D4632.F  ; 出料開爪原點燈_15
D4633.5  ; 出料托框回流原點燈_5
D4633.6  ; 出料托框回流原點燈_6
D4633.7  ; 出料托框回流原點燈_7
D4633.8  ; 出料托框回流原點燈_8
D4633.9  ; 出料托框回流原點燈_9
D4633.A  ; 出料托框回流原點燈_10
D4633.B  ; 出料托框回流原點燈_11
D4633.C  ; 出料托框回流原點燈_12
D4633.D  ; 出料托框回流原點燈_13
D4633.E  ; 出料托框回流原點燈_14
D4633.F  ; 出料托框回流原點燈_15
D4634.5  ; 出料手臂原點燈_5
D4634.6  ; 出料手臂原點燈_6
D4634.7  ; 出料手臂原點燈_7
D4634.8  ; 出料手臂原點燈_8
D4634.9  ; 出料手臂原點燈_9
D4634.A  ; 出料手臂原點燈_10
D4634.B  ; 出料手臂原點燈_11
D4634.C  ; 出料手臂原點燈_12
D4634.D  ; 出料手臂原點燈_13
D4634.E  ; 出料手臂原點燈_14
D4634.F  ; 出料手臂原點燈_15
D4635.4  ; 出料牙叉原點燈_4
D4635.5  ; 出料牙叉原點燈_5
D4635.6  ; 出料牙叉原點燈_6
D4635.7  ; 出料牙叉原點燈_7
D4635.8  ; 出料牙叉原點燈_8
D4635.9  ; 出料牙叉原點燈_9
D4635.A  ; 出料牙叉原點燈_10
D4635.B  ; 出料牙叉原點燈_11
D4635.C  ; 出料牙叉原點燈_12
D4635.D  ; 出料牙叉原點燈_13
D4635.E  ; 出料牙叉原點燈_14
D4635.F  ; 出料牙叉原點燈_15
D9450.0  ; 重要異常
D9450.1  ; 馬達異常
D9450.2  ; 馬達極限異常
D9450.3  ; 氣缸異常
D9450.4  ; 掉框板異常
D9450.5  ; 安全門異常
D9450.6  ; 光電異常
D9450.7  ; EGO 超溫異常數量
D9450.8  ; 風車異常數量
D9450.9  ; 超溫異常數量
D9450.A  ; 低溫異常數量
D9450.B  ; ELB 跳脫異常數量
D9451.0  ; 熱風低溫異常
D9451.1  ; ELB 跳脫異常
D9451.2  ; 伺服马达不在位置上異常
D9451.6  ; 輸送馬達逾時
D9451.7  ; 輸送馬達無歸零要求
D9452.0  ; IRA EGO超溫異常數量
D9452.1  ; IRA 超溫異常數量
D9452.2  ; IRA 低溫異常數量
D9452.3  ; IRB EGO超溫異常數量
D9452.4  ; IRB 超溫異常數量
D9452.5  ; IRB 低溫異常數量
D9452.6  ; SCR異常數量
